LIN {X 0,Y 204.503,Z 1254.176,A -85,B 0,C 180,E1 10684.827,E2 10684.827} C_VEL
LIN {X 0,Y 208.439,Z 1245.49,A -85,B 0,C 180,E1 10678.799,E2 10678.799} C_VEL
LIN {X 0,Y 214.044,Z 1235.485,A -85,B 0,C 180,E1 10673.28,E2 10673.28} C_VEL
LIN {X 0,Y 221.45,Z 1223.468,A -85,B 0,C 180,E1 10668.071,E2 10668.071} C_VEL
LIN {X 0,Y 230.083,Z 1210.068,A -85,B 0,C 180,E1 10663.473,E2 10663.473} C_VEL
LIN {X 0,Y 239.593,Z 1195.363,A -85,B 0,C 180,E1 10659.465,E2 10659.465} C_VEL
LIN {X 0,Y 249.64,Z 1179.288,A -85,B 0,C 180,E1 10655.999,E2 10655.999} C_VEL
LIN {X 0,Y 259.481,Z 1162.559,A -85,B 0,C 180,E1 10653.172,E2 10653.172} C_VEL
LIN {X 0,Y 269.687,Z 1143.852,A -85,B 0,C 180,E1 10650.671,E2 10650.671} C_VEL
LIN {X 0,Y 279.054,Z 1124.999,A -85,B 0,C 180,E1 10648.693,E2 10648.693} C_VEL
LIN {X 0,Y 287.565,Z 1105.557,A -85,B 0,C 180,E1 10647.117,E2 10647.117} C_VEL
LIN {X 0,Y 295.468,Z 1084.875,A -85,B 0,C 180,E1 10645.827,E2 10645.827} C_VEL
LIN {X 0,Y 302.047,Z 1064.618,A -85,B 0,C 180,E1 10644.86,E2 10644.86} C_VEL
LIN {X 0,Y 307.636,Z 1042.346,A -85,B 0,C 180,E1 10644.026,E2 10644.026} C_VEL
LIN {X 0,Y 311.673,Z 1019.917,A -85,B 0,C 180,E1 10643.369,E2 10643.369} C_VEL
LIN {X 0,Y 314.482,Z 994.588,A -85,B 0,C 180,E1 10642.797,E2 10642.797} C_VEL
LIN {X 0,Y 326.356,Z 856.623,A -85,B 0,C 180,E1 10640.021,E2 10640.021} C_VEL
LIN {X 0,Y 321.509,Z 844.673,A -85,B 0,C 180,E1 10636.857,E2 10636.857} C_VEL
LIN {X 0,Y 317.747,Z 835.882,A -85,B 0,C 180,E1 10633.929,E2 10633.929} C_VEL
LIN {X 0,Y 314.507,Z 828.3,A -85,B 0,C 180,E1 10630.79,E2 10630.79} C_VEL
LIN {X 0,Y 311.943,Z 822.087,A -85,B 0,C 180,E1 10627.458,E2 10627.458} C_VEL
LIN {X 0,Y 310.729,Z 819.454,A -85,B 0,C 180,E1 10625.354,E2 10625.354} C_VEL
LIN {X 0,Y 308.92,Z 817.37,A -85,B 0,C 180,E1 10619.072,E2 10619.072} C_VEL
LIN {X 0,Y 309.517,Z 818.382,A -85,B 0,C 180,E1 10614.81,E2 10614.81} C_VEL
LIN {X 0,Y 310.912,Z 819.791,A -85,B 0,C 180,E1 10611.772,E2 10611.772} C_VEL
LIN {X 0,Y 313.909,Z 824.972,A -85,B 0,C 180,E1 10607.584,E2 10607.584} C_VEL
LIN {X 0,Y 316.917,Z 830.011,A -85,B 0,C 180,E1 10604.632,E2 10604.632} C_VEL
LIN {X 0,Y 320.006,Z 835.239,A -85,B 0,C 180,E1 10602.169,E2 10602.169} C_VEL
LIN {X 0,Y 324.529,Z 843.076,A -85,B 0,C 180,E1 10599.154,E2 10599.154} C_VEL
LIN {X 0,Y 326.398,Z 846.717,A -85,B 0,C 180,E1 10598.029,E2 10598.029} C_VEL
LIN {X 0,Y 316.958,Z 955.602,A -85,B 0,C 180,E1 10595.822,E2 10595.822} C_VEL
LIN {X 0,Y 314.556,Z 977.677,A -85,B 0,C 180,E1 10595.158,E2 10595.158} C_VEL
LIN {X 0,Y 310.815,Z 999.575,A -85,B 0,C 180,E1 10594.26,E2 10594.26} C_VEL
LIN {X 0,Y 306.147,Z 1019.787,A -85,B 0,C 180,E1 10593.187,E2 10593.187} C_VEL
LIN {X 0,Y 300.378,Z 1039.215,A -85,B 0,C 180,E1 10591.893,E2 10591.893} C_VEL
LIN {X 0,Y 293.495,Z 1058.383,A -85,B 0,C 180,E1 10590.307,E2 10590.307} C_VEL
LIN {X 0,Y 285.739,Z 1076.805,A -85,B 0,C 180,E1 10588.433,E2 10588.433} C_VEL
LIN {X 0,Y 277.363,Z 1093.945,A -85,B 0,C 180,E1 10586.278,E2 10586.278} C_VEL
LIN {X 0,Y 268.375,Z 1110.195,A -85,B 0,C 180,E1 10583.762,E2 10583.762} C_VEL
LIN {X 0,Y 259.092,Z 1125.356,A -85,B 0,C 180,E1 10580.864,E2 10580.864} C_VEL
LIN {X 0,Y 250.087,Z 1138.686,A -85,B 0,C 180,E1 10577.699,E2 10577.699} C_VEL
LIN {X 0,Y 240.767,Z 1151.437,A -85,B 0,C 180,E1 10573.908,E2 10573.908} C_VEL
LIN {X 0,Y 231.962,Z 1162.798,A -85,B 0,C 180,E1 10569.637,E2 10569.637} C_VEL
LIN {X 0,Y 223.916,Z 1172.716,A -85,B 0,C 180,E1 10564.858,E2 10564.858} C_VEL
LIN {X 0,Y 216.928,Z 1181.075,A -85,B 0,C 180,E1 10559.549,E2 10559.549} C_VEL
LIN {X 0,Y 211.256,Z 1187.948,A -85,B 0,C 180,E1 10553.721,E2 10553.721} C_VEL
LIN {X 0,Y 207.413,Z 1192.886,A -85,B 0,C 180,E1 10547.969,E2 10547.969} C_VEL
LIN {X 0,Y 204.994,Z 1196.234,A -85,B 0,C 180,E1 10542.106,E2 10542.106} C_VEL
LIN {X 0,Y 203.675,Z 1198.296,A -85,B 0,C 180,E1 10535.917,E2 10535.917} C_VEL
LIN {X 0,Y 203.338,Z 1198.982,A -85,B 0,C 180,E1 10530.282,E2 10530.282} C_VEL
LIN {X 0,Y 203.603,Z 1198.438,A -85,B 0,C 180,E1 10524.646,E2 10524.646} C_VEL
LIN {X 0,Y 204.744,Z 1196.714,A -85,B 0,C 180,E1 10518.736,E2 10518.736} C_VEL
LIN {X 0,Y 207.077,Z 1193.329,A -85,B 0,C 180,E1 10512.581,E2 10512.581} C_VEL
LIN {X 0,Y 210.986,Z 1188.339,A -85,B 0,C 180,E1 10506.543,E2 10506.543} C_VEL
LIN {X 0,Y 216.415,Z 1181.796,A -85,B 0,C 180,E1 10500.834,E2 10500.834} C_VEL
LIN {X 0,Y 223.321,Z 1173.527,A -85,B 0,C 180,E1 10495.469,E2 10495.469} C_VEL
LIN {X 0,Y 231.054,Z 1164.004,A -85,B 0,C 180,E1 10490.769,E2 10490.769} C_VEL
LIN {X 0,Y 240.16,Z 1152.37,A -85,B 0,C 180,E1 10486.284,E2 10486.284} C_VEL
LIN {X 0,Y 249.432,Z 1139.816,A -85,B 0,C 180,E1 10482.477,E2 10482.477} C_VEL
LIN {X 0,Y 258.967,Z 1125.723,A -85,B 0,C 180,E1 10479.102,E2 10479.102} C_VEL
LIN {X 0,Y 268.247,Z 1110.632,A -85,B 0,C 180,E1 10476.201,E2 10476.201} C_VEL
LIN {X 0,Y 277.137,Z 1094.668,A -85,B 0,C 180,E1 10473.711,E2 10473.711} C_VEL
LIN {X 0,Y 285.608,Z 1077.369,A -85,B 0,C 180,E1 10471.524,E2 10471.524} C_VEL
LIN {X 0,Y 293.368,Z 1059.066,A -85,B 0,C 180,E1 10469.65,E2 10469.65} C_VEL
LIN {X 0,Y 300.496,Z 1039.32,A -85,B 0,C 180,E1 10468.01,E2 10468.01} C_VEL
LIN {X 0,Y 306.179,Z 1020.196,A -85,B 0,C 180,E1 10466.733,E2 10466.733} C_VEL
LIN {X 0,Y 311.012,Z 999.341,A -85,B 0,C 180,E1 10465.626,E2 10465.626} C_VEL
LIN {X 0,Y 314.792,Z 977.037,A -85,B 0,C 180,E1 10464.718,E2 10464.718} C_VEL
LIN {X 0,Y 317.162,Z 954.96,A -85,B 0,C 180,E1 10464.06,E2 10464.06} C_VEL
LIN {X 0,Y 326.534,Z 846.621,A -85,B 0,C 180,E1 10461.851,E2 10461.851} C_VEL
LIN {X 0,Y 321.954,Z 838.389,A -85,B 0,C 180,E1 10458.985,E2 10458.985} C_VEL
LIN {X 0,Y 318.029,Z 831.737,A -85,B 0,C 180,E1 10456.062,E2 10456.062} C_VEL
LIN {X 0,Y 315.638,Z 827.791,A -85,B 0,C 180,E1 10453.931,E2 10453.931} C_VEL
LIN {X 0,Y 313.48,Z 824.081,A -85,B 0,C 180,E1 10451.592,E2 10451.592} C_VEL
LIN {X 0,Y 312.025,Z 822.099,A -85,B 0,C 180,E1 10449.716,E2 10449.716} C_VEL
LIN {X 0,Y 311.103,Z 821.621,A -85,B 0,C 180,E1 10448.407,E2 10448.407} C_VEL
LIN {X 0,Y 309.694,Z 823.43,A -85,B 0,C 180,E1 10446.383,E2 10446.383} C_VEL
LIN {X 0,Y 308.511,Z 825.827,A -85,B 0,C 180,E1 10444.02,E2 10444.02} C_VEL
LIN {X 0,Y 308.312,Z 825.919,A -85,B 0,C 180,E1 10443.183,E2 10443.183} C_VEL
LIN {X 0,Y 308.242,Z 825.769,A -85,B 0,C 180,E1 10439.814,E2 10439.814} C_VEL
LIN {X 0,Y 309.952,Z 827.753,A -85,B 0,C 180,E1 10434.632,E2 10434.632} C_VEL
LIN {X 0,Y 311.302,Z 831.115,A -85,B 0,C 180,E1 10432.248,E2 10432.248} C_VEL
LIN {X 0,Y 313.701,Z 836.931,A -85,B 0,C 180,E1 10429.161,E2 10429.161} C_VEL
LIN {X 0,Y 317.548,Z 846.48,A -85,B 0,C 180,E1 10425.457,E2 10425.457} C_VEL
LIN {X 0,Y 321.377,Z 856.081,A -85,B 0,C 180,E1 10422.529,E2 10422.529} C_VEL
LIN {X 0,Y 323.306,Z 861.466,A -85,B 0,C 180,E1 10421.198,E2 10421.198} C_VEL
LIN {X 0,Y 309.794,Z 1010.819,A -85,B 0,C 180,E1 10418.218,E2 10418.218} C_VEL
LIN {X 0,Y 306.147,Z 1033.255,A -85,B 0,C 180,E1 10417.618,E2 10417.618} C_VEL
LIN {X 0,Y 300.877,Z 1055.874,A -85,B 0,C 180,E1 10416.851,E2 10416.851} C_VEL
LIN {X 0,Y 294.479,Z 1076.961,A -85,B 0,C 180,E1 10415.956,E2 10415.956} C_VEL
LIN {X 0,Y 286.773,Z 1097.528,A -85,B 0,C 180,E1 10414.812,E2 10414.812} C_VEL
LIN {X 0,Y 278.03,Z 1117.659,A -85,B 0,C 180,E1 10413.333,E2 10413.333} C_VEL
LIN {X 0,Y 268.525,Z 1137.044,A -85,B 0,C 180,E1 10411.489,E2 10411.489} C_VEL
LIN {X 0,Y 258.368,Z 1155.588,A -85,B 0,C 180,E1 10409.215,E2 10409.215} C_VEL
LIN {X 0,Y 248.104,Z 1172.667,A -85,B 0,C 180,E1 10406.531,E2 10406.531} C_VEL
LIN {X 0,Y 237.325,Z 1189.476,A -85,B 0,C 180,E1 10403.173,E2 10403.173} C_VEL
LIN {X 0,Y 227.365,Z 1204.365,A -85,B 0,C 180,E1 10399.395,E2 10399.395} C_VEL
LIN {X 0,Y 217.967,Z 1218.039,A -85,B 0,C 180,E1 10394.943,E2 10394.943} C_VEL
LIN {X 0,Y 209.514,Z 1230.606,A -85,B 0,C 180,E1 10389.752,E2 10389.752} C_VEL
LIN {X 0,Y 202.783,Z 1241.437,A -85,B 0,C 180,E1 10384.071,E2 10384.071} C_VEL
LIN {X 0,Y 197.975,Z 1250.46,A -85,B 0,C 180,E1 10378.013,E2 10378.013} C_VEL
LIN {X 0,Y 195.11,Z 1257.789,A -85,B 0,C 180,E1 10371.651,E2 10371.651} C_VEL
LIN {X 0,Y 194.074,Z 1263.415,A -85,B 0,C 180,E1 10365.233,E2 10365.233} C_VEL
LIN {X 0,Y 194.355,Z 1266.89,A -85,B 0,C 180,E1 10359.475,E2 10359.475} C_VEL
LIN {X 0,Y 195.05,Z 1268.792,A -85,B 0,C 180,E1 10354.41,E2 10354.41} C_VEL
LIN {X 0,Y 195.396,Z 1269.368,A -85,B 0,C 180,E1 10350,E2 10350} C_VEL
LIN {X 0,Y 195.051,Z 1268.784,A -85,B 0,C 180,E1 10345.59,E2 10345.59} C_VEL
LIN {X 0,Y 194.358,Z 1266.876,A -85,B 0,C 180,E1 10340.525,E2 10340.525} C_VEL
LIN {X 0,Y 194.075,Z 1263.395,A -85,B 0,C 180,E1 10334.767,E2 10334.767} C_VEL
LIN {X 0,Y 195.111,Z 1257.763,A -85,B 0,C 180,E1 10328.349,E2 10328.349} C_VEL
LIN {X 0,Y 197.976,Z 1250.423,A -85,B 0,C 180,E1 10321.987,E2 10321.987} C_VEL
LIN {X 0,Y 202.888,Z 1241.215,A -85,B 0,C 180,E1 10315.82,E2 10315.82} C_VEL
LIN {X 0,Y 209.622,Z 1230.376,A -85,B 0,C 180,E1 10310.169,E2 10310.169} C_VEL
LIN {X 0,Y 218.43,Z 1217.266,A -85,B 0,C 180,E1 10304.807,E2 10304.807} C_VEL
LIN {X 0,Y 227.549,Z 1203.98,A -85,B 0,C 180,E1 10300.523,E2 10300.523} C_VEL
LIN {X 0,Y 237.811,Z 1188.63,A -85,B 0,C 180,E1 10296.657,E2 10296.657} C_VEL
LIN {X 0,Y 248.097,Z 1172.525,A -85,B 0,C 180,E1 10293.467,E2 10293.467} C_VEL
LIN {X 0,Y 258.358,Z 1155.409,A -85,B 0,C 180,E1 10290.782,E2 10290.782} C_VEL
LIN {X 0,Y 268.135,Z 1137.555,A -85,B 0,C 180,E1 10288.587,E2 10288.587} C_VEL
LIN {X 0,Y 277.633,Z 1118.248,A -85,B 0,C 180,E1 10286.733,E2 10286.733} C_VEL
LIN {X 0,Y 286.322,Z 1098.341,A -85,B 0,C 180,E1 10285.255,E2 10285.255} C_VEL
LIN {X 0,Y 294.117,Z 1077.571,A -85,B 0,C 180,E1 10284.089,E2 10284.089} C_VEL
LIN {X 0,Y 300.513,Z 1056.674,A -85,B 0,C 180,E1 10283.193,E2 10283.193} C_VEL
LIN {X 0,Y 305.922,Z 1033.657,A -85,B 0,C 180,E1 10282.406,E2 10282.406} C_VEL
LIN {X 0,Y 309.597,Z 1011.199,A -85,B 0,C 180,E1 10281.803,E2 10281.803} C_VEL
LIN {X 0,Y 321.287,Z 881.947,A -85,B 0,C 180,E1 10279.213,E2 10279.213} C_VEL
LIN {X 0,Y 323.122,Z 860.936,A -85,B 0,C 180,E1 10278.772,E2 10278.772} C_VEL
LIN {X 0,Y 318.787,Z 849.865,A -85,B 0,C 180,E1 10275.695,E2 10275.695} C_VEL
LIN {X 0,Y 315.749,Z 842.456,A -85,B 0,C 180,E1 10273.132,E2 10273.132} C_VEL
LIN {X 0,Y 312.944,Z 835.521,A -85,B 0,C 180,E1 10270.214,E2 10270.214} C_VEL
LIN {X 0,Y 310.65,Z 829.666,A -85,B 0,C 180,E1 10267.025,E2 10267.025} C_VEL
LIN {X 0,Y 309.548,Z 827.277,A -85,B 0,C 180,E1 10265.003,E2 10265.003} C_VEL
LIN {X 0,Y 307.943,Z 825.297,A -85,B 0,C 180,E1 10258.883,E2 10258.883} C_VEL
LIN {X 0,Y 308.882,Z 826.716,A -85,B 0,C 180,E1 10253.868,E2 10253.868} C_VEL
LIN {X 0,Y 309.825,Z 827.75,A -85,B 0,C 180,E1 10251.93,E2 10251.93} C_VEL
LIN {X 0,Y 312.678,Z 832.844,A -85,B 0,C 180,E1 10247.816,E2 10247.816} C_VEL
LIN {X 0,Y 315.421,Z 837.566,A -85,B 0,C 180,E1 10245.028,E2 10245.028} C_VEL
LIN {X 0,Y 319.312,Z 844.257,A -85,B 0,C 180,E1 10241.893,E2 10241.893} C_VEL
LIN {X 0,Y 323.211,Z 851.495,A -85,B 0,C 180,E1 10239.265,E2 10239.265} C_VEL
LIN {X 0,Y 313.851,Z 956.436,A -85,B 0,C 180,E1 10237.152,E2 10237.152} C_VEL
LIN {X 0,Y 311.402,Z 978.497,A -85,B 0,C 180,E1 10236.496,E2 10236.496} C_VEL
LIN {X 0,Y 307.529,Z 1000.715,A -85,B 0,C 180,E1 10235.595,E2 10235.595} C_VEL
LIN {X 0,Y 302.837,Z 1020.632,A -85,B 0,C 180,E1 10234.552,E2 10234.552} C_VEL
LIN {X 0,Y 296.748,Z 1040.612,A -85,B 0,C 180,E1 10233.235,E2 10233.235} C_VEL
LIN {X 0,Y 289.672,Z 1059.779,A -85,B 0,C 180,E1 10231.661,E2 10231.661} C_VEL
LIN {X 0,Y 281.69,Z 1078.201,A -85,B 0,C 180,E1 10229.8,E2 10229.8} C_VEL
LIN {X 0,Y 272.902,Z 1095.643,A -85,B 0,C 180,E1 10227.616,E2 10227.616} C_VEL
LIN {X 0,Y 263.781,Z 1111.586,A -85,B 0,C 180,E1 10225.149,E2 10225.149} C_VEL
LIN {X 0,Y 254.167,Z 1126.757,A -85,B 0,C 180,E1 10222.249,E2 10222.249} C_VEL
LIN {X 0,Y 244.817,Z 1140.088,A -85,B 0,C 180,E1 10219.072,E2 10219.072} C_VEL
LIN {X 0,Y 235.107,Z 1152.841,A -85,B 0,C 180,E1 10215.251,E2 10215.251} C_VEL
LIN {X 0,Y 225.891,Z 1164.204,A -85,B 0,C 180,E1 10210.925,E2 10210.925} C_VEL
LIN {X 0,Y 217.427,Z 1174.123,A -85,B 0,C 180,E1 10206.058,E2 10206.058} C_VEL
LIN {X 0,Y 210.035,Z 1182.482,A -85,B 0,C 180,E1 10200.621,E2 10200.621} C_VEL
LIN {X 0,Y 203.992,Z 1189.354,A -85,B 0,C 180,E1 10194.621,E2 10194.621} C_VEL
LIN {X 0,Y 199.876,Z 1194.288,A -85,B 0,C 180,E1 10188.672,E2 10188.672} C_VEL
LIN {X 0,Y 197.258,Z 1197.632,A -85,B 0,C 180,E1 10182.589,E2 10182.589} C_VEL
LIN {X 0,Y 195.826,Z 1199.688,A -85,B 0,C 180,E1 10176.155,E2 10176.155} C_VEL
LIN {X 0,Y 195.461,Z 1200.373,A -85,B 0,C 180,E1 10170.293,E2 10170.293} C_VEL
LIN {X 0,Y 195.749,Z 1199.829,A -85,B 0,C 180,E1 10164.431,E2 10164.431} C_VEL
LIN {X 0,Y 196.987,Z 1198.11,A -85,B 0,C 180,E1 10158.286,E2 10158.286} C_VEL
LIN {X 0,Y 199.511,Z 1194.73,A -85,B 0,C 180,E1 10151.898,E2 10151.898} C_VEL
LIN {X 0,Y 203.706,Z 1189.743,A -85,B 0,C 180,E1 10145.651,E2 10145.651} C_VEL
LIN {X 0,Y 209.345,Z 1183.378,A -85,B 0,C 180,E1 10139.902,E2 10139.902} C_VEL
LIN {X 0,Y 216.567,Z 1175.187,A -85,B 0,C 180,E1 10134.429,E2 10134.429} C_VEL
LIN {X 0,Y 224.875,Z 1165.489,A -85,B 0,C 180,E1 10129.523,E2 10129.523} C_VEL
LIN {X 0,Y 234.479,Z 1153.771,A -85,B 0,C 180,E1 10124.941,E2 10124.941} C_VEL
LIN {X 0,Y 244.143,Z 1141.214,A -85,B 0,C 180,E1 10121.103,E2 10121.103} C_VEL
LIN {X 0,Y 254.043,Z 1127.119,A -85,B 0,C 180,E1 10117.715,E2 10117.715} C_VEL
LIN {X 0,Y 263.651,Z 1112.025,A -85,B 0,C 180,E1 10114.813,E2 10114.813} C_VEL
LIN {X 0,Y 272.698,Z 1096.316,A -85,B 0,C 180,E1 10112.366,E2 10112.366} C_VEL
LIN {X 0,Y 281.564,Z 1078.757,A -85,B 0,C 180,E1 10110.156,E2 10110.156} C_VEL
LIN {X 0,Y 289.549,Z 1060.452,A -85,B 0,C 180,E1 10108.294,E2 10108.294} C_VEL
LIN {X 0,Y 296.635,Z 1041.453,A -85,B 0,C 180,E1 10106.722,E2 10106.722} C_VEL
LIN {X 0,Y 302.716,Z 1021.58,A -85,B 0,C 180,E1 10105.401,E2 10105.401} C_VEL
LIN {X 0,Y 307.685,Z 1000.721,A -85,B 0,C 180,E1 10104.302,E2 10104.302} C_VEL
LIN {X 0,Y 311.574,Z 978.414,A -85,B 0,C 180,E1 10103.399,E2 10103.399} C_VEL
LIN {X 0,Y 314.022,Z 956.329,A -85,B 0,C 180,E1 10102.743,E2 10102.743} C_VEL
LIN {X 0,Y 323.31,Z 851.467,A -85,B 0,C 180,E1 10100.597,E2 10100.597} C_VEL
LIN {X 0,Y 319.054,Z 843.692,A -85,B 0,C 180,E1 10097.697,E2 10097.697} C_VEL
LIN {X 0,Y 315.502,Z 837.537,A -85,B 0,C 180,E1 10094.781,E2 10094.781} C_VEL
LIN {X 0,Y 312.197,Z 831.799,A -85,B 0,C 180,E1 10091.266,E2 10091.266} C_VEL
LIN {X 0,Y 309.761,Z 827.402,A -85,B 0,C 180,E1 10087.419,E2 10087.419} C_VEL
LIN {X 0,Y 308.312,Z 825.919,A -85,B 0,C 180,E1 10083.183,E2 10083.183} C_VEL
LIN {X 0,Y 308.071,Z 826.562,A -85,B 0,C 180,E1 10081.851,E2 10081.851} C_VEL
LIN {X 0,Y 307.707,Z 830.18,A -85,B 0,C 180,E1 10079.77,E2 10079.77} C_VEL
LIN {X 0,Y 307.754,Z 834.066,A -85,B 0,C 180,E1 10077.574,E2 10077.574} C_VEL
LIN {X 0,Y 307.988,Z 834.719,A -85,B 0,C 180,E1 10076.748,E2 10076.748} C_VEL
LIN {X 0,Y 308.868,Z 835.69,A -85,B 0,C 180,E1 10074.8,E2 10074.8} C_VEL
LIN {X 0,Y 310.059,Z 838.814,A -85,B 0,C 180,E1 10072.589,E2 10072.589} C_VEL
LIN {X 0,Y 312.272,Z 844.511,A -85,B 0,C 180,E1 10069.578,E2 10069.578} C_VEL
LIN {X 0,Y 315.763,Z 853.626,A -85,B 0,C 180,E1 10066.029,E2 10066.029} C_VEL
LIN {X 0,Y 319.367,Z 863.118,A -85,B 0,C 180,E1 10063.12,E2 10063.12} C_VEL
LIN {X 0,Y 320.243,Z 865.843,A -85,B 0,C 180,E1 10062.46,E2 10062.46} C_VEL
LIN {X 0,Y 306.873,Z 1009.439,A -85,B 0,C 180,E1 10059.624,E2 10059.624} C_VEL
LIN {X 0,Y 303.144,Z 1031.872,A -85,B 0,C 180,E1 10059.035,E2 10059.035} C_VEL
LIN {X 0,Y 297.613,Z 1055.051,A -85,B 0,C 180,E1 10058.263,E2 10058.263} C_VEL
LIN {X 0,Y 291.047,Z 1076.14,A -85,B 0,C 180,E1 10057.384,E2 10057.384} C_VEL
LIN {X 0,Y 283.113,Z 1096.815,A -85,B 0,C 180,E1 10056.259,E2 10056.259} C_VEL
LIN {X 0,Y 274.051,Z 1117.051,A -85,B 0,C 180,E1 10054.794,E2 10054.794} C_VEL
LIN {X 0,Y 264.54,Z 1135.858,A -85,B 0,C 180,E1 10053.029,E2 10053.029} C_VEL
LIN {X 0,Y 254.108,Z 1154.319,A -85,B 0,C 180,E1 10050.797,E2 10050.797} C_VEL
LIN {X 0,Y 243.602,Z 1171.198,A -85,B 0,C 180,E1 10048.168,E2 10048.168} C_VEL
LIN {X 0,Y 232.395,Z 1187.998,A -85,B 0,C 180,E1 10044.829,E2 10044.829} C_VEL
LIN {X 0,Y 222.179,Z 1202.598,A -85,B 0,C 180,E1 10041.125,E2 10041.125} C_VEL
LIN {X 0,Y 212.561,Z 1215.854,A -85,B 0,C 180,E1 10036.809,E2 10036.809} C_VEL
LIN {X 0,Y 203.49,Z 1228.54,A -85,B 0,C 180,E1 10031.553,E2 10031.553} C_VEL
LIN {X 0,Y 196.282,Z 1239.311,A -85,B 0,C 180,E1 10025.859,E2 10025.859} C_VEL
LIN {X 0,Y 190.815,Z 1248.57,A -85,B 0,C 180,E1 10019.508,E2 10019.508} C_VEL
LIN {X 0,Y 187.422,Z 1256.269,A -85,B 0,C 180,E1 10012.645,E2 10012.645} C_VEL
LIN {X 0,Y 186.158,Z 1261.965,A -85,B 0,C 180,E1 10005.897,E2 10005.897} C_VEL
LIN {X 0,Y 186.395,Z 1265.465,A -85,B 0,C 180,E1 9999.884,E2 9999.884} C_VEL
LIN {X 0,Y 187.128,Z 1267.39,A -85,B 0,C 180,E1 9994.597,E2 9994.597} C_VEL
LIN {X 0,Y 187.517,Z 1267.978,A -85,B 0,C 180,E1 9990,E2 9990} C_VEL
LIN {X 0,Y 187.129,Z 1267.382,A -85,B 0,C 180,E1 9985.403,E2 9985.403} C_VEL
LIN {X 0,Y 186.397,Z 1265.451,A -85,B 0,C 180,E1 9980.116,E2 9980.116} C_VEL
LIN {X 0,Y 186.165,Z 1261.892,A -85,B 0,C 180,E1 9974.021,E2 9974.021} C_VEL
LIN {X 0,Y 187.425,Z 1256.24,A -85,B 0,C 180,E1 9967.353,E2 9967.353} C_VEL
LIN {X 0,Y 190.815,Z 1248.53,A -85,B 0,C 180,E1 9960.492,E2 9960.492} C_VEL
LIN {X 0,Y 196.374,Z 1239.116,A -85,B 0,C 180,E1 9954.053,E2 9954.053} C_VEL
LIN {X 0,Y 203.899,Z 1227.901,A -85,B 0,C 180,E1 9948.173,E2 9948.173} C_VEL
LIN {X 0,Y 213.053,Z 1215.077,A -85,B 0,C 180,E1 9942.939,E2 9942.939} C_VEL
LIN {X 0,Y 222.974,Z 1201.339,A -85,B 0,C 180,E1 9938.557,E2 9938.557} C_VEL
LIN {X 0,Y 233.655,Z 1186.075,A -85,B 0,C 180,E1 9934.757,E2 9934.757} C_VEL
LIN {X 0,Y 244.282,Z 1169.981,A -85,B 0,C 180,E1 9931.644,E2 9931.644} C_VEL
LIN {X 0,Y 255.67,Z 1151.401,A -85,B 0,C 180,E1 9928.839,E2 9928.839} C_VEL
LIN {X 0,Y 265.833,Z 1133.253,A -85,B 0,C 180,E1 9926.714,E2 9926.714} C_VEL
LIN {X 0,Y 275.331,Z 1114.112,A -85,B 0,C 180,E1 9924.984,E2 9924.984} C_VEL
LIN {X 0,Y 284.178,Z 1093.822,A -85,B 0,C 180,E1 9923.577,E2 9923.577} C_VEL
LIN {X 0,Y 291.704,Z 1073.828,A -85,B 0,C 180,E1 9922.524,E2 9922.524} C_VEL
LIN {X 0,Y 298.327,Z 1051.97,A -85,B 0,C 180,E1 9921.633,E2 9921.633} C_VEL
LIN {X 0,Y 303.385,Z 1029.836,A -85,B 0,C 180,E1 9920.918,E2 9920.918} C_VEL
LIN {X 0,Y 307.012,Z 1006.706,A -85,B 0,C 180,E1 9920.33,E2 9920.33} C_VEL
LIN {X 0,Y 320.098,Z 865.479,A -85,B 0,C 180,E1 9917.543,E2 9917.543} C_VEL
LIN {X 0,Y 316.451,Z 855.814,A -85,B 0,C 180,E1 9914.735,E2 9914.735} C_VEL
LIN {X 0,Y 313.905,Z 849.247,A -85,B 0,C 180,E1 9912.415,E2 9912.415} C_VEL
LIN {X 0,Y 311.398,Z 842.697,A -85,B 0,C 180,E1 9909.611,E2 9909.611} C_VEL
LIN {X 0,Y 309.321,Z 837.129,A -85,B 0,C 180,E1 9906.496,E2 9906.496} C_VEL
LIN {X 0,Y 308.476,Z 835.166,A -85,B 0,C 180,E1 9904.834,E2 9904.834} C_VEL
LIN {X 0,Y 306.968,Z 833.238,A -85,B 0,C 180,E1 9898.88,E2 9898.88} C_VEL
LIN {X 0,Y 307.987,Z 834.758,A -85,B 0,C 180,E1 9893.663,E2 9893.663} C_VEL
LIN {X 0,Y 308.74,Z 835.704,A -85,B 0,C 180,E1 9892.089,E2 9892.089} C_VEL
LIN {X 0,Y 311.379,Z 840.551,A -85,B 0,C 180,E1 9888.14,E2 9888.14} C_VEL
LIN {X 0,Y 313.94,Z 845.121,A -85,B 0,C 180,E1 9885.427,E2 9885.427} C_VEL
LIN {X 0,Y 317.591,Z 851.642,A -85,B 0,C 180,E1 9882.361,E2 9882.361} C_VEL
LIN {X 0,Y 320.145,Z 856.609,A -85,B 0,C 180,E1 9880.519,E2 9880.519} C_VEL
LIN {X 0,Y 310.931,Z 957.084,A -85,B 0,C 180,E1 9878.513,E2 9878.513} C_VEL
LIN {X 0,Y 308.435,Z 979.222,A -85,B 0,C 180,E1 9877.864,E2 9877.864} C_VEL
LIN {X 0,Y 304.425,Z 1001.803,A -85,B 0,C 180,E1 9876.961,E2 9876.961} C_VEL
LIN {X 0,Y 299.536,Z 1022.031,A -85,B 0,C 180,E1 9875.912,E2 9875.912} C_VEL
LIN {X 0,Y 293.285,Z 1042.009,A -85,B 0,C 180,E1 9874.609,E2 9874.609} C_VEL
LIN {X 0,Y 286.016,Z 1061.175,A -85,B 0,C 180,E1 9873.05,E2 9873.05} C_VEL
LIN {X 0,Y 278.163,Z 1078.893,A -85,B 0,C 180,E1 9871.286,E2 9871.286} C_VEL
LIN {X 0,Y 269.096,Z 1096.403,A -85,B 0,C 180,E1 9869.124,E2 9869.124} C_VEL
LIN {X 0,Y 259.304,Z 1113.046,A -85,B 0,C 180,E1 9866.573,E2 9866.573} C_VEL
LIN {X 0,Y 249.395,Z 1128.157,A -85,B 0,C 180,E1 9863.689,E2 9863.689} C_VEL
LIN {X 0,Y 239.695,Z 1141.491,A -85,B 0,C 180,E1 9860.505,E2 9860.505} C_VEL
LIN {X 0,Y 229.583,Z 1154.245,A -85,B 0,C 180,E1 9856.659,E2 9856.659} C_VEL
LIN {X 0,Y 219.937,Z 1165.611,A -85,B 0,C 180,E1 9852.284,E2 9852.284} C_VEL
LIN {X 0,Y 211.042,Z 1175.53,A -85,B 0,C 180,E1 9847.33,E2 9847.33} C_VEL
LIN {X 0,Y 203.222,Z 1183.889,A -85,B 0,C 180,E1 9841.764,E2 9841.764} C_VEL
LIN {X 0,Y 196.782,Z 1190.76,A -85,B 0,C 180,E1 9835.587,E2 9835.587} C_VEL
LIN {X 0,Y 192.37,Z 1195.69,A -85,B 0,C 180,E1 9829.429,E2 9829.429} C_VEL
LIN {X 0,Y 189.44,Z 1199.166,A -85,B 0,C 180,E1 9822.807,E2 9822.807} C_VEL
LIN {X 0,Y 187.982,Z 1201.081,A -85,B 0,C 180,E1 9816.413,E2 9816.413} C_VEL
LIN {X 0,Y 187.583,Z 1201.763,A -85,B 0,C 180,E1 9810.305,E2 9810.305} C_VEL
LIN {X 0,Y 187.899,Z 1201.222,A -85,B 0,C 180,E1 9804.197,E2 9804.197} C_VEL
LIN {X 0,Y 189.241,Z 1199.507,A -85,B 0,C 180,E1 9797.799,E2 9797.799} C_VEL
LIN {X 0,Y 191.98,Z 1196.131,A -85,B 0,C 180,E1 9791.162,E2 9791.162} C_VEL
LIN {X 0,Y 196.479,Z 1191.147,A -85,B 0,C 180,E1 9784.694,E2 9784.694} C_VEL
LIN {X 0,Y 202.49,Z 1184.783,A -85,B 0,C 180,E1 9778.771,E2 9778.771} C_VEL
LIN {X 0,Y 210.136,Z 1176.591,A -85,B 0,C 180,E1 9773.165,E2 9773.165} C_VEL
LIN {X 0,Y 218.882,Z 1166.891,A -85,B 0,C 180,E1 9768.171,E2 9768.171} C_VEL
LIN {X 0,Y 228.933,Z 1155.172,A -85,B 0,C 180,E1 9763.533,E2 9763.533} C_VEL
LIN {X 0,Y 239,Z 1142.612,A -85,B 0,C 180,E1 9759.669,E2 9759.669} C_VEL
LIN {X 0,Y 249.274,Z 1128.514,A -85,B 0,C 180,E1 9756.274,E2 9756.274} C_VEL
LIN {X 0,Y 259.214,Z 1113.418,A -85,B 0,C 180,E1 9753.377,E2 9753.377} C_VEL
LIN {X 0,Y 268.977,Z 1096.908,A -85,B 0,C 180,E1 9750.834,E2 9750.834} C_VEL
LIN {X 0,Y 278.04,Z 1079.44,A -85,B 0,C 180,E1 9748.667,E2 9748.667} C_VEL
LIN {X 0,Y 286.26,Z 1060.97,A -85,B 0,C 180,E1 9746.825,E2 9746.825} C_VEL
LIN {X 0,Y 293.905,Z 1040.648,A -85,B 0,C 180,E1 9745.19,E2 9745.19} C_VEL
LIN {X 0,Y 299.979,Z 1021.05,A -85,B 0,C 180,E1 9743.926,E2 9743.926} C_VEL
LIN {X 0,Y 305.031,Z 999.773,A -85,B 0,C 180,E1 9742.843,E2 9742.843} C_VEL
LIN {X 0,Y 308.766,Z 978.042,A -85,B 0,C 180,E1 9741.995,E2 9741.995} C_VEL
LIN {X 0,Y 311.314,Z 954.493,A -85,B 0,C 180,E1 9741.321,E2 9741.321} C_VEL
LIN {X 0,Y 320.308,Z 856.643,A -85,B 0,C 180,E1 9739.375,E2 9739.375} C_VEL
LIN {X 0,Y 316.455,Z 849.501,A -85,B 0,C 180,E1 9736.521,E2 9736.521} C_VEL
LIN {X 0,Y 313.032,Z 843.311,A -85,B 0,C 180,E1 9733.39,E2 9733.39} C_VEL
LIN {X 0,Y 310.778,Z 839.337,A -85,B 0,C 180,E1 9730.755,E2 9730.755} C_VEL
LIN {X 0,Y 308.598,Z 835.224,A -85,B 0,C 180,E1 9727.073,E2 9727.073} C_VEL
LIN {X 0,Y 307.197,Z 833.534,A -85,B 0,C 180,E1 9721.306,E2 9721.306} C_VEL
LIN {X 0,Y 307.988,Z 834.719,A -85,B 0,C 180,E1 9716.748,E2 9716.748} C_VEL
LIN {X 0,Y 308.381,Z 836.177,A -85,B 0,C 180,E1 9715.548,E2 9715.548} C_VEL
LIN {X 0,Y 308.782,Z 840.188,A -85,B 0,C 180,E1 9714.067,E2 9714.067} C_VEL
LIN {X 0,Y 309.737,Z 848.626,A -85,B 0,C 180,E1 9711.557,E2 9711.557} C_VEL
LIN {X 0,Y 310.244,Z 850.455,A -85,B 0,C 180,E1 9710.791,E2 9710.791} C_VEL
LIN {X 0,Y 313.234,Z 858.526,A -85,B 0,C 180,E1 9707.37,E2 9707.37} C_VEL
LIN {X 0,Y 316.665,Z 868.171,A -85,B 0,C 180,E1 9704.291,E2 9704.291} C_VEL
LIN {X 0,Y 317.334,Z 870.262,A -85,B 0,C 180,E1 9703.744,E2 9703.744} C_VEL
LIN {X 0,Y 304.142,Z 1008.043,A -85,B 0,C 180,E1 9701.056,E2 9701.056} C_VEL
LIN {X 0,Y 300.337,Z 1030.453,A -85,B 0,C 180,E1 9700.48,E2 9700.48} C_VEL
LIN {X 0,Y 294.706,Z 1053.629,A -85,B 0,C 180,E1 9699.728,E2 9699.728} C_VEL
LIN {X 0,Y 288.274,Z 1074.055,A -85,B 0,C 180,E1 9698.904,E2 9698.904} C_VEL
LIN {X 0,Y 280.186,Z 1094.768,A -85,B 0,C 180,E1 9697.821,E2 9697.821} C_VEL
LIN {X 0,Y 271.074,Z 1114.778,A -85,B 0,C 180,E1 9696.429,E2 9696.429} C_VEL
LIN {X 0,Y 261.453,Z 1133.451,A -85,B 0,C 180,E1 9694.743,E2 9694.743} C_VEL
LIN {X 0,Y 251.032,Z 1151.398,A -85,B 0,C 180,E1 9692.645,E2 9692.645} C_VEL
LIN {X 0,Y 239.679,Z 1169.171,A -85,B 0,C 180,E1 9689.961,E2 9689.961} C_VEL
LIN {X 0,Y 228.325,Z 1185.619,A -85,B 0,C 180,E1 9686.76,E2 9686.76} C_VEL
LIN {X 0,Y 217.6,Z 1200.288,A -85,B 0,C 180,E1 9683.082,E2 9683.082} C_VEL
LIN {X 0,Y 207.397,Z 1213.67,A -85,B 0,C 180,E1 9678.768,E2 9678.768} C_VEL
LIN {X 0,Y 197.688,Z 1226.477,A -85,B 0,C 180,E1 9673.459,E2 9673.459} C_VEL
LIN {X 0,Y 189.848,Z 1237.33,A -85,B 0,C 180,E1 9667.655,E2 9667.655} C_VEL
LIN {X 0,Y 183.785,Z 1246.678,A -85,B 0,C 180,E1 9661.119,E2 9661.119} C_VEL
LIN {X 0,Y 179.862,Z 1254.544,A -85,B 0,C 180,E1 9653.941,E2 9653.941} C_VEL
LIN {X 0,Y 178.292,Z 1260.307,A -85,B 0,C 180,E1 9646.954,E2 9646.954} C_VEL
LIN {X 0,Y 178.399,Z 1263.886,A -85,B 0,C 180,E1 9640.658,E2 9640.658} C_VEL
LIN {X 0,Y 179.158,Z 1265.895,A -85,B 0,C 180,E1 9635.123,E2 9635.123} C_VEL
LIN {X 0,Y 179.621,Z 1266.544,A -85,B 0,C 180,E1 9630.638,E2 9630.638} C_VEL
LIN {X 0,Y 179.345,Z 1266.197,A -85,B 0,C 180,E1 9626.164,E2 9626.164} C_VEL
LIN {X 0,Y 178.538,Z 1264.475,A -85,B 0,C 180,E1 9620.654,E2 9620.654} C_VEL
LIN {X 0,Y 178.203,Z 1261.323,A -85,B 0,C 180,E1 9614.71,E2 9614.71} C_VEL
LIN {X 0,Y 179.407,Z 1255.747,A -85,B 0,C 180,E1 9607.385,E2 9607.385} C_VEL
LIN {X 0,Y 182.666,Z 1248.656,A -85,B 0,C 180,E1 9600.487,E2 9600.487} C_VEL
LIN {X 0,Y 188.2,Z 1239.617,A -85,B 0,C 180,E1 9593.855,E2 9593.855} C_VEL
LIN {X 0,Y 195.956,Z 1228.706,A -85,B 0,C 180,E1 9587.662,E2 9587.662} C_VEL
LIN {X 0,Y 204.81,Z 1217.061,A -85,B 0,C 180,E1 9582.512,E2 9582.512} C_VEL
LIN {X 0,Y 215.269,Z 1203.249,A -85,B 0,C 180,E1 9577.813,E2 9577.813} C_VEL
LIN {X 0,Y 226.354,Z 1188.201,A -85,B 0,C 180,E1 9573.859,E2 9573.859} C_VEL
LIN {X 0,Y 237.372,Z 1172.499,A -85,B 0,C 180,E1 9570.642,E2 9570.642} C_VEL
LIN {X 0,Y 248.03,Z 1156.091,A -85,B 0,C 180,E1 9568.017,E2 9568.017} C_VEL
LIN {X 0,Y 258.697,Z 1138.078,A -85,B 0,C 180,E1 9565.774,E2 9565.774} C_VEL
LIN {X 0,Y 268.626,Z 1119.513,A -85,B 0,C 180,E1 9563.971,E2 9563.971} C_VEL
LIN {X 0,Y 277.665,Z 1100.293,A -85,B 0,C 180,E1 9562.539,E2 9562.539} C_VEL
LIN {X 0,Y 285.69,Z 1080.552,A -85,B 0,C 180,E1 9561.422,E2 9561.422} C_VEL
LIN {X 0,Y 292.986,Z 1059.117,A -85,B 0,C 180,E1 9560.488,E2 9560.488} C_VEL
LIN {X 0,Y 298.823,Z 1036.922,A -85,B 0,C 180,E1 9559.721,E2 9559.721} C_VEL
LIN {X 0,Y 302.97,Z 1014.751,A -85,B 0,C 180,E1 9559.116,E2 9559.116} C_VEL
LIN {X 0,Y 306.279,Z 985.823,A -85,B 0,C 180,E1 9558.501,E2 9558.501} C_VEL
LIN {X 0,Y 317.165,Z 869.887,A -85,B 0,C 180,E1 9556.247,E2 9556.247} C_VEL
LIN {X 0,Y 313.689,Z 860.215,A -85,B 0,C 180,E1 9553.267,E2 9553.267} C_VEL
LIN {X 0,Y 310.45,Z 851.308,A -85,B 0,C 180,E1 9549.734,E2 9549.734} C_VEL
LIN {X 0,Y 308.223,Z 845.041,A -85,B 0,C 180,E1 9546.332,E2 9546.332} C_VEL
LIN {X 0,Y 307.405,Z 843.055,A -85,B 0,C 180,E1 9544.664,E2 9544.664} C_VEL
LIN {X 0,Y 305.993,Z 841.179,A -85,B 0,C 180,E1 9538.876,E2 9538.876} C_VEL
LIN {X 0,Y 307.096,Z 842.801,A -85,B 0,C 180,E1 9533.456,E2 9533.456} C_VEL
LIN {X 0,Y 307.659,Z 843.649,A -85,B 0,C 180,E1 9532.249,E2 9532.249} C_VEL
LIN {X 0,Y 310.09,Z 848.257,A -85,B 0,C 180,E1 9528.468,E2 9528.468} C_VEL
LIN {X 0,Y 312.565,Z 852.855,A -85,B 0,C 180,E1 9525.74,E2 9525.74} C_VEL
LIN {X 0,Y 315.947,Z 859.143,A -85,B 0,C 180,E1 9522.789,E2 9522.789} C_VEL
LIN {X 0,Y 317.223,Z 861.85,A -85,B 0,C 180,E1 9521.794,E2 9521.794} C_VEL
LIN {X 0,Y 308.179,Z 957.865,A -85,B 0,C 180,E1 9519.896,E2 9519.896} C_VEL
LIN {X 0,Y 305.595,Z 980.312,A -85,B 0,C 180,E1 9519.245,E2 9519.245} C_VEL
LIN {X 0,Y 301.439,Z 1003.159,A -85,B 0,C 180,E1 9518.342,E2 9518.342} C_VEL
LIN {X 0,Y 296.408,Z 1023.429,A -85,B 0,C 180,E1 9517.302,E2 9517.302} C_VEL
LIN {X 0,Y 289.995,Z 1043.406,A -85,B 0,C 180,E1 9516.015,E2 9516.015} C_VEL
LIN {X 0,Y 282.531,Z 1062.571,A -85,B 0,C 180,E1 9514.475,E2 9514.475} C_VEL
LIN {X 0,Y 274.461,Z 1080.289,A -85,B 0,C 180,E1 9512.731,E2 9512.731} C_VEL
LIN {X 0,Y 265.13,Z 1097.801,A -85,B 0,C 180,E1 9510.589,E2 9510.589} C_VEL
LIN {X 0,Y 255.407,Z 1113.865,A -85,B 0,C 180,E1 9508.155,E2 9508.155} C_VEL
LIN {X 0,Y 245.438,Z 1128.686,A -85,B 0,C 180,E1 9505.374,E2 9505.374} C_VEL
LIN {X 0,Y 234.729,Z 1142.894,A -85,B 0,C 180,E1 9502,E2 9502} C_VEL
LIN {X 0,Y 224.206,Z 1155.649,A -85,B 0,C 180,E1 9498.135,E2 9498.135} C_VEL
LIN {X 0,Y 214.116,Z 1167.017,A -85,B 0,C 180,E1 9493.717,E2 9493.717} C_VEL
LIN {X 0,Y 204.767,Z 1176.937,A -85,B 0,C 180,E1 9488.682,E2 9488.682} C_VEL
LIN {X 0,Y 196.495,Z 1185.296,A -85,B 0,C 180,E1 9482.987,E2 9482.987} C_VEL
LIN {X 0,Y 189.632,Z 1192.166,A -85,B 0,C 180,E1 9476.626,E2 9476.626} C_VEL
LIN {X 0,Y 184.902,Z 1197.092,A -85,B 0,C 180,E1 9470.247,E2 9470.247} C_VEL
LIN {X 0,Y 181.725,Z 1200.565,A -85,B 0,C 180,E1 9463.361,E2 9463.361} C_VEL
LIN {X 0,Y 180.142,Z 1202.474,A -85,B 0,C 180,E1 9456.693,E2 9456.693} C_VEL
LIN {X 0,Y 179.704,Z 1203.153,A -85,B 0,C 180,E1 9450.319,E2 9450.319} C_VEL
LIN {X 0,Y 180.05,Z 1202.614,A -85,B 0,C 180,E1 9443.944,E2 9443.944} C_VEL
LIN {X 0,Y 181.509,Z 1200.904,A -85,B 0,C 180,E1 9437.271,E2 9437.271} C_VEL
LIN {X 0,Y 184.483,Z 1197.531,A -85,B 0,C 180,E1 9430.366,E2 9430.366} C_VEL
LIN {X 0,Y 189.31,Z 1192.552,A -85,B 0,C 180,E1 9423.664,E2 9423.664} C_VEL
LIN {X 0,Y 195.722,Z 1186.188,A -85,B 0,C 180,E1 9417.562,E2 9417.562} C_VEL
LIN {X 0,Y 203.816,Z 1177.996,A -85,B 0,C 180,E1 9411.823,E2 9411.823} C_VEL
LIN {X 0,Y 213.016,Z 1168.294,A -85,B 0,C 180,E1 9406.743,E2 9406.743} C_VEL
LIN {X 0,Y 223.534,Z 1156.572,A -85,B 0,C 180,E1 9402.056,E2 9402.056} C_VEL
LIN {X 0,Y 234.014,Z 1144.01,A -85,B 0,C 180,E1 9398.173,E2 9398.173} C_VEL
LIN {X 0,Y 244.67,Z 1129.91,A -85,B 0,C 180,E1 9394.777,E2 9394.777} C_VEL
LIN {X 0,Y 254.857,Z 1114.951,A -85,B 0,C 180,E1 9391.916,E2 9391.916} C_VEL
LIN {X 0,Y 264.665,Z 1098.934,A -85,B 0,C 180,E1 9389.453,E2 9389.453} C_VEL
LIN {X 0,Y 273.976,Z 1081.533,A -85,B 0,C 180,E1 9387.301,E2 9387.301} C_VEL
LIN {X 0,Y 282.417,Z 1063.223,A -85,B 0,C 180,E1 9385.476,E2 9385.476} C_VEL
LIN {X 0,Y 289.89,Z 1044.22,A -85,B 0,C 180,E1 9383.939,E2 9383.939} C_VEL
LIN {X 0,Y 296.299,Z 1024.343,A -85,B 0,C 180,E1 9382.647,E2 9382.647} C_VEL
LIN {X 0,Y 301.525,Z 1003.545,A -85,B 0,C 180,E1 9381.574,E2 9381.574} C_VEL
LIN {X 0,Y 305.63,Z 981.302,A -85,B 0,C 180,E1 9380.687,E2 9380.687} C_VEL
LIN {X 0,Y 308.234,Z 959.318,A -85,B 0,C 180,E1 9380.038,E2 9380.038} C_VEL
LIN {X 0,Y 314.756,Z 889.383,A -85,B 0,C 180,E1 9378.626,E2 9378.626} C_VEL
LIN {X 0,Y 317.377,Z 861.724,A -85,B 0,C 180,E1 9378.078,E2 9378.078} C_VEL
LIN {X 0,Y 313.502,Z 854.385,A -85,B 0,C 180,E1 9374.877,E2 9374.877} C_VEL
LIN {X 0,Y 311.273,Z 850.331,A -85,B 0,C 180,E1 9372.617,E2 9372.617} C_VEL
LIN {X 0,Y 309.522,Z 847.049,A -85,B 0,C 180,E1 9370.422,E2 9370.422} C_VEL
LIN {X 0,Y 307.536,Z 843.115,A -85,B 0,C 180,E1 9366.909,E2 9366.909} C_VEL
LIN {X 0,Y 306.222,Z 841.479,A -85,B 0,C 180,E1 9361.123,E2 9361.123} C_VEL
LIN {X 0,Y 307.674,Z 843.247,A -85,B 0,C 180,E1 9355.247,E2 9355.247} C_VEL
LIN {X 0,Y 308.827,Z 846.511,A -85,B 0,C 180,E1 9352.933,E2 9352.933} C_VEL
LIN {X 0,Y 310.244,Z 850.455,A -85,B 0,C 180,E1 9350.791,E2 9350.791} C_VEL
LIN {X 0,Y 311.002,Z 853.48,A -85,B 0,C 180,E1 9349.709,E2 9349.709} C_VEL
LIN {X 0,Y 311.872,Z 859.853,A -85,B 0,C 180,E1 9348.29,E2 9348.29} C_VEL
LIN {X 0,Y 313.394,Z 870.6,A -85,B 0,C 180,E1 9346.171,E2 9346.171} C_VEL
LIN {X 0,Y 313.896,Z 872.538,A -85,B 0,C 180,E1 9345.671,E2 9345.671} C_VEL
LIN {X 0,Y 314.561,Z 874.93,A -85,B 0,C 180,E1 9345.048,E2 9345.048} C_VEL
LIN {X 0,Y 301.593,Z 1006.741,A -85,B 0,C 180,E1 9342.512,E2 9342.512} C_VEL
LIN {X 0,Y 297.706,Z 1029.126,A -85,B 0,C 180,E1 9341.95,E2 9341.95} C_VEL
LIN {X 0,Y 292.038,Z 1052.059,A -85,B 0,C 180,E1 9341.227,E2 9341.227} C_VEL
LIN {X 0,Y 285.457,Z 1072.631,A -85,B 0,C 180,E1 9340.422,E2 9340.422} C_VEL
LIN {X 0,Y 277.218,Z 1093.339,A -85,B 0,C 180,E1 9339.378,E2 9339.378} C_VEL
LIN {X 0,Y 267.907,Z 1113.339,A -85,B 0,C 180,E1 9338.033,E2 9338.033} C_VEL
LIN {X 0,Y 258.154,Z 1131.826,A -85,B 0,C 180,E1 9336.414,E2 9336.414} C_VEL
LIN {X 0,Y 247.338,Z 1149.941,A -85,B 0,C 180,E1 9334.348,E2 9334.348} C_VEL
LIN {X 0,Y 235.972,Z 1167.195,A -85,B 0,C 180,E1 9331.801,E2 9331.801} C_VEL
LIN {X 0,Y 224.528,Z 1183.241,A -85,B 0,C 180,E1 9328.757,E2 9328.757} C_VEL
LIN {X 0,Y 213.254,Z 1198.016,A -85,B 0,C 180,E1 9325.11,E2 9325.11} C_VEL
LIN {X 0,Y 202.419,Z 1211.592,A -85,B 0,C 180,E1 9320.783,E2 9320.783} C_VEL
LIN {X 0,Y 192.589,Z 1223.837,A -85,B 0,C 180,E1 9315.76,E2 9315.76} C_VEL
LIN {X 0,Y 183.986,Z 1234.804,A -85,B 0,C 180,E1 9309.885,E2 9309.885} C_VEL
LIN {X 0,Y 177.162,Z 1244.37,A -85,B 0,C 180,E1 9303.191,E2 9303.191} C_VEL
LIN {X 0,Y 172.707,Z 1252.142,A -85,B 0,C 180,E1 9296.102,E2 9296.102} C_VEL
LIN {X 0,Y 170.554,Z 1258.106,A -85,B 0,C 180,E1 9288.809,E2 9288.809} C_VEL
LIN {X 0,Y 170.393,Z 1262.303,A -85,B 0,C 180,E1 9281.496,E2 9281.496} C_VEL
LIN {X 0,Y 171.105,Z 1264.297,A -85,B 0,C 180,E1 9276.038,E2 9276.038} C_VEL
LIN {X 0,Y 171.687,Z 1265.065,A -85,B 0,C 180,E1 9271.669,E2 9271.669} C_VEL
LIN {X 0,Y 171.661,Z 1265.03,A -85,B 0,C 180,E1 9267.997,E2 9267.997} C_VEL
LIN {X 0,Y 171.045,Z 1264.18,A -85,B 0,C 180,E1 9263.586,E2 9263.586} C_VEL
LIN {X 0,Y 170.338,Z 1261.971,A -85,B 0,C 180,E1 9257.801,E2 9257.801} C_VEL
LIN {X 0,Y 170.671,Z 1257.564,A -85,B 0,C 180,E1 9250.493,E2 9250.493} C_VEL
LIN {X 0,Y 173.023,Z 1251.486,A -85,B 0,C 180,E1 9243.209,E2 9243.209} C_VEL
LIN {X 0,Y 177.708,Z 1243.501,A -85,B 0,C 180,E1 9236.152,E2 9236.152} C_VEL
LIN {X 0,Y 184.755,Z 1233.704,A -85,B 0,C 180,E1 9229.504,E2 9229.504} C_VEL
LIN {X 0,Y 193.551,Z 1222.56,A -85,B 0,C 180,E1 9223.681,E2 9223.681} C_VEL
LIN {X 0,Y 204.121,Z 1209.43,A -85,B 0,C 180,E1 9218.468,E2 9218.468} C_VEL
LIN {X 0,Y 215.187,Z 1195.376,A -85,B 0,C 180,E1 9214.204,E2 9214.204} C_VEL
LIN {X 0,Y 227.106,Z 1179.545,A -85,B 0,C 180,E1 9210.501,E2 9210.501} C_VEL
LIN {X 0,Y 238.947,Z 1162.757,A -85,B 0,C 180,E1 9207.492,E2 9207.492} C_VEL
LIN {X 0,Y 249.677,Z 1145.94,A -85,B 0,C 180,E1 9205.175,E2 9205.175} C_VEL
LIN {X 0,Y 260.885,Z 1126.549,A -85,B 0,C 180,E1 9203.105,E2 9203.105} C_VEL
LIN {X 0,Y 270.421,Z 1108.053,A -85,B 0,C 180,E1 9201.586,E2 9201.586} C_VEL
LIN {X 0,Y 278.934,Z 1088.893,A -85,B 0,C 180,E1 9200.391,E2 9200.391} C_VEL
LIN {X 0,Y 287.194,Z 1067.042,A -85,B 0,C 180,E1 9199.361,E2 9199.361} C_VEL
LIN {X 0,Y 293.724,Z 1045.48,A -85,B 0,C 180,E1 9198.557,E2 9198.557} C_VEL
LIN {X 0,Y 298.724,Z 1023.257,A -85,B 0,C 180,E1 9197.901,E2 9197.901} C_VEL
LIN {X 0,Y 302.124,Z 1000.655,A -85,B 0,C 180,E1 9197.373,E2 9197.373} C_VEL
LIN {X 0,Y 314.376,Z 874.467,A -85,B 0,C 180,E1 9194.928,E2 9194.928} C_VEL
LIN {X 0,Y 311.236,Z 865.2,A -85,B 0,C 180,E1 9191.911,E2 9191.911} C_VEL
LIN {X 0,Y 308.663,Z 857.777,A -85,B 0,C 180,E1 9188.757,E2 9188.757} C_VEL
LIN {X 0,Y 306.882,Z 852.387,A -85,B 0,C 180,E1 9185.703,E2 9185.703} C_VEL
LIN {X 0,Y 306.248,Z 850.875,A -85,B 0,C 180,E1 9184.306,E2 9184.306} C_VEL
LIN {X 0,Y 305.019,Z 849.113,A -85,B 0,C 180,E1 9178.685,E2 9178.685} C_VEL
LIN {X 0,Y 306.389,Z 850.992,A -85,B 0,C 180,E1 9172.876,E2 9172.876} C_VEL
LIN {X 0,Y 308.812,Z 855.962,A -85,B 0,C 180,E1 9168.798,E2 9168.798} C_VEL
LIN {X 0,Y 311.2,Z 860.586,A -85,B 0,C 180,E1 9166.056,E2 9166.056} C_VEL
LIN {X 0,Y 314.472,Z 866.965,A -85,B 0,C 180,E1 9163.095,E2 9163.095} C_VEL
LIN {X 0,Y 305.604,Z 958.707,A -85,B 0,C 180,E1 9161.302,E2 9161.302} C_VEL
LIN {X 0,Y 302.936,Z 981.403,A -85,B 0,C 180,E1 9160.651,E2 9160.651} C_VEL
LIN {X 0,Y 298.75,Z 1003.989,A -85,B 0,C 180,E1 9159.773,E2 9159.773} C_VEL
LIN {X 0,Y 293.459,Z 1024.828,A -85,B 0,C 180,E1 9158.721,E2 9158.721} C_VEL
LIN {X 0,Y 286.883,Z 1044.803,A -85,B 0,C 180,E1 9157.452,E2 9157.452} C_VEL
LIN {X 0,Y 278.973,Z 1064.544,A -85,B 0,C 180,E1 9155.884,E2 9155.884} C_VEL
LIN {X 0,Y 270.187,Z 1083.095,A -85,B 0,C 180,E1 9154.056,E2 9154.056} C_VEL
LIN {X 0,Y 260.621,Z 1100.473,A -85,B 0,C 180,E1 9151.928,E2 9151.928} C_VEL
LIN {X 0,Y 250.623,Z 1116.318,A -85,B 0,C 180,E1 9149.508,E2 9149.508} C_VEL
LIN {X 0,Y 239.682,Z 1131.831,A -85,B 0,C 180,E1 9146.542,E2 9146.542} C_VEL
LIN {X 0,Y 228.68,Z 1145.879,A -85,B 0,C 180,E1 9143.14,E2 9143.14} C_VEL
LIN {X 0,Y 217.822,Z 1158.356,A -85,B 0,C 180,E1 9139.233,E2 9139.233} C_VEL
LIN {X 0,Y 207.391,Z 1169.477,A -85,B 0,C 180,E1 9134.738,E2 9134.738} C_VEL
LIN {X 0,Y 197.705,Z 1179.22,A -85,B 0,C 180,E1 9129.584,E2 9129.584} C_VEL
LIN {X 0,Y 189.122,Z 1187.432,A -85,B 0,C 180,E1 9123.718,E2 9123.718} C_VEL
LIN {X 0,Y 182.266,Z 1193.839,A -85,B 0,C 180,E1 9117.438,E2 9117.438} C_VEL
LIN {X 0,Y 177.065,Z 1198.849,A -85,B 0,C 180,E1 9110.493,E2 9110.493} C_VEL
LIN {X 0,Y 173.811,Z 1202.236,A -85,B 0,C 180,E1 9103.303,E2 9103.303} C_VEL
LIN {X 0,Y 172.211,Z 1203.979,A -85,B 0,C 180,E1 9096.333,E2 9096.333} C_VEL
LIN {X 0,Y 171.826,Z 1204.553,A -85,B 0,C 180,E1 9089.667,E2 9089.667} C_VEL
LIN {X 0,Y 172.296,Z 1203.895,A -85,B 0,C 180,E1 9083,E2 9083} C_VEL
LIN {X 0,Y 174.117,Z 1201.893,A -85,B 0,C 180,E1 9075.705,E2 9075.705} C_VEL
LIN {X 0,Y 177.628,Z 1198.401,A -85,B 0,C 180,E1 9068.539,E2 9068.539} C_VEL
LIN {X 0,Y 183.073,Z 1193.154,A -85,B 0,C 180,E1 9061.632,E2 9061.632} C_VEL
LIN {X 0,Y 190.545,Z 1186.133,A -85,B 0,C 180,E1 9055.114,E2 9055.114} C_VEL
LIN {X 0,Y 198.978,Z 1178.075,A -85,B 0,C 180,E1 9049.594,E2 9049.594} C_VEL
LIN {X 0,Y 208.86,Z 1168.117,A -85,B 0,C 180,E1 9044.498,E2 9044.498} C_VEL
LIN {X 0,Y 218.875,Z 1157.32,A -85,B 0,C 180,E1 9040.283,E2 9040.283} C_VEL
LIN {X 0,Y 229.82,Z 1144.615,A -85,B 0,C 180,E1 9036.405,E2 9036.405} C_VEL
LIN {X 0,Y 240.238,Z 1131.305,A -85,B 0,C 180,E1 9033.225,E2 9033.225} C_VEL
LIN {X 0,Y 250.966,Z 1116.041,A -85,B 0,C 180,E1 9030.33,E2 9030.33} C_VEL
LIN {X 0,Y 261.4,Z 1099.391,A -85,B 0,C 180,E1 9027.818,E2 9027.818} C_VEL
LIN {X 0,Y 270.825,Z 1082.216,A -85,B 0,C 180,E1 9025.737,E2 9025.737} C_VEL
LIN {X 0,Y 279.499,Z 1063.741,A -85,B 0,C 180,E1 9023.939,E2 9023.939} C_VEL
LIN {X 0,Y 287.551,Z 1043.415,A -85,B 0,C 180,E1 9022.348,E2 9022.348} C_VEL
LIN {X 0,Y 294.094,Z 1023.242,A -85,B 0,C 180,E1 9021.086,E2 9021.086} C_VEL
LIN {X 0,Y 299.383,Z 1002.005,A -85,B 0,C 180,E1 9020.036,E2 9020.036} C_VEL
LIN {X 0,Y 303.271,Z 980.365,A -85,B 0,C 180,E1 9019.214,E2 9019.214} C_VEL
LIN {X 0,Y 306.029,Z 955.996,A -85,B 0,C 180,E1 9018.532,E2 9018.532} C_VEL
LIN {X 0,Y 314.597,Z 866.992,A -85,B 0,C 180,E1 9016.764,E2 9016.764} C_VEL
LIN {X 0,Y 311.383,Z 860.733,A -85,B 0,C 180,E1 9013.841,E2 9013.841} C_VEL
LIN {X 0,Y 308.617,Z 855.21,A -85,B 0,C 180,E1 9010.548,E2 9010.548} C_VEL
LIN {X 0,Y 306.476,Z 851.006,A -85,B 0,C 180,E1 9006.745,E2 9006.745} C_VEL
LIN {X 0,Y 305.247,Z 849.419,A -85,B 0,C 180,E1 9001.126,E2 9001.126} C_VEL
LIN {X 0,Y 306.563,Z 851.074,A -85,B 0,C 180,E1 8995.511,E2 8995.511} C_VEL
LIN {X 0,Y 307.657,Z 854.366,A -85,B 0,C 180,E1 8993.188,E2 8993.188} C_VEL
LIN {X 0,Y 309.605,Z 860.087,A -85,B 0,C 180,E1 8990.239,E2 8990.239} C_VEL
LIN {X 0,Y 312.29,Z 867.915,A -85,B 0,C 180,E1 8987.19,E2 8987.19} C_VEL
LIN {X 0,Y 313.896,Z 872.538,A -85,B 0,C 180,E1 8985.671,E2 8985.671} C_VEL
LIN {X 0,Y 314.067,Z 874.595,A -85,B 0,C 180,E1 8985.389,E2 8985.389} C_VEL
LIN {X 0,Y 313.78,Z 877.976,A -85,B 0,C 180,E1 8985.296,E2 8985.296} C_VEL
LIN {X 0,Y 312.688,Z 883.798,A -85,B 0,C 180,E1 8985.522,E2 8985.522} C_VEL
LIN {X 0,Y 310.753,Z 892.768,A -85,B 0,C 180,E1 8986.05,E2 8986.05} C_VEL
LIN {X 0,Y 310.289,Z 896.165,A -85,B 0,C 180,E1 8986.071,E2 8986.071} C_VEL
LIN {X 0,Y 299.216,Z 1005.655,A -85,B 0,C 180,E1 8983.987,E2 8983.987} C_VEL
LIN {X 0,Y 295.204,Z 1028.143,A -85,B 0,C 180,E1 8983.434,E2 8983.434} C_VEL
LIN {X 0,Y 289.442,Z 1050.934,A -85,B 0,C 180,E1 8982.736,E2 8982.736} C_VEL
LIN {X 0,Y 282.399,Z 1072.355,A -85,B 0,C 180,E1 8981.919,E2 8981.919} C_VEL
LIN {X 0,Y 274.46,Z 1091.91,A -85,B 0,C 180,E1 8980.967,E2 8980.967} C_VEL
LIN {X 0,Y 265,Z 1111.818,A -85,B 0,C 180,E1 8979.679,E2 8979.679} C_VEL
LIN {X 0,Y 254.868,Z 1130.555,A -85,B 0,C 180,E1 8978.09,E2 8978.09} C_VEL
LIN {X 0,Y 243.873,Z 1148.486,A -85,B 0,C 180,E1 8976.1,E2 8976.1} C_VEL
LIN {X 0,Y 231.937,Z 1166.037,A -85,B 0,C 180,E1 8973.56,E2 8973.56} C_VEL
LIN {X 0,Y 219.588,Z 1182.667,A -85,B 0,C 180,E1 8970.419,E2 8970.419} C_VEL
LIN {X 0,Y 207.74,Z 1197.565,A -85,B 0,C 180,E1 8966.724,E2 8966.724} C_VEL
LIN {X 0,Y 196.439,Z 1210.998,A -85,B 0,C 180,E1 8962.354,E2 8962.354} C_VEL
LIN {X 0,Y 185.218,Z 1224.15,A -85,B 0,C 180,E1 8956.72,E2 8956.72} C_VEL
LIN {X 0,Y 176.118,Z 1235.156,A -85,B 0,C 180,E1 8950.471,E2 8950.471} C_VEL
LIN {X 0,Y 169.043,Z 1244.533,A -85,B 0,C 180,E1 8943.371,E2 8943.371} C_VEL
LIN {X 0,Y 164.581,Z 1251.908,A -85,B 0,C 180,E1 8935.938,E2 8935.938} C_VEL
LIN {X 0,Y 162.528,Z 1257.605,A -85,B 0,C 180,E1 8928.285,E2 8928.285} C_VEL
LIN {X 0,Y 162.483,Z 1261.173,A -85,B 0,C 180,E1 8921.356,E2 8921.356} C_VEL
LIN {X 0,Y 163.321,Z 1263.173,A -85,B 0,C 180,E1 8915.269,E2 8915.269} C_VEL
LIN {X 0,Y 163.858,Z 1263.763,A -85,B 0,C 180,E1 8910.699,E2 8910.699} C_VEL
LIN {X 0,Y 163.608,Z 1263.482,A -85,B 0,C 180,E1 8906.496,E2 8906.496} C_VEL
LIN {X 0,Y 162.676,Z 1261.923,A -85,B 0,C 180,E1 8900.448,E2 8900.448} C_VEL
LIN {X 0,Y 162.377,Z 1258.628,A -85,B 0,C 180,E1 8893.546,E2 8893.546} C_VEL
LIN {X 0,Y 163.879,Z 1253.422,A -85,B 0,C 180,E1 8885.873,E2 8885.873} C_VEL
LIN {X 0,Y 167.75,Z 1246.411,A -85,B 0,C 180,E1 8878.365,E2 8878.365} C_VEL
LIN {X 0,Y 174.113,Z 1237.579,A -85,B 0,C 180,E1 8871.25,E2 8871.25} C_VEL
LIN {X 0,Y 182.867,Z 1226.871,A -85,B 0,C 180,E1 8864.702,E2 8864.702} C_VEL
LIN {X 0,Y 193.226,Z 1214.74,A -85,B 0,C 180,E1 8859.09,E2 8859.09} C_VEL
LIN {X 0,Y 204.045,Z 1201.865,A -85,B 0,C 180,E1 8854.593,E2 8854.593} C_VEL
LIN {X 0,Y 216.755,Z 1186.138,A -85,B 0,C 180,E1 8850.393,E2 8850.393} C_VEL
LIN {X 0,Y 228.746,Z 1170.364,A -85,B 0,C 180,E1 8847.192,E2 8847.192} C_VEL
LIN {X 0,Y 240.681,Z 1153.156,A -85,B 0,C 180,E1 8844.528,E2 8844.528} C_VEL
LIN {X 0,Y 252.005,Z 1135.09,A -85,B 0,C 180,E1 8842.388,E2 8842.388} C_VEL
LIN {X 0,Y 262.818,Z 1115.778,A -85,B 0,C 180,E1 8840.635,E2 8840.635} C_VEL
LIN {X 0,Y 272.41,Z 1096.187,A -85,B 0,C 180,E1 8839.289,E2 8839.289} C_VEL
LIN {X 0,Y 280.755,Z 1076.165,A -85,B 0,C 180,E1 8838.264,E2 8838.264} C_VEL
LIN {X 0,Y 288.371,Z 1053.985,A -85,B 0,C 180,E1 8837.382,E2 8837.382} C_VEL
LIN {X 0,Y 294.29,Z 1031.724,A -85,B 0,C 180,E1 8836.674,E2 8836.674} C_VEL
LIN {X 0,Y 298.478,Z 1009.225,A -85,B 0,C 180,E1 8836.106,E2 8836.106} C_VEL
LIN {X 0,Y 302.112,Z 976.85,A -85,B 0,C 180,E1 8835.458,E2 8835.458} C_VEL
LIN {X 0,Y 311.763,Z 879.008,A -85,B 0,C 180,E1 8833.588,E2 8833.588} C_VEL
LIN {X 0,Y 309.236,Z 871.33,A -85,B 0,C 180,E1 8830.903,E2 8830.903} C_VEL
LIN {X 0,Y 307.142,Z 864.768,A -85,B 0,C 180,E1 8828.046,E2 8828.046} C_VEL
LIN {X 0,Y 305.58,Z 859.722,A -85,B 0,C 180,E1 8825.068,E2 8825.068} C_VEL
LIN {X 0,Y 305.186,Z 858.764,A -85,B 0,C 180,E1 8824.133,E2 8824.133} C_VEL
LIN {X 0,Y 304.044,Z 857.054,A -85,B 0,C 180,E1 8818.681,E2 8818.681} C_VEL
LIN {X 0,Y 305.323,Z 858.911,A -85,B 0,C 180,E1 8813.04,E2 8813.04} C_VEL
LIN {X 0,Y 307.609,Z 863.82,A -85,B 0,C 180,E1 8809.038,E2 8809.038} C_VEL
LIN {X 0,Y 309.845,Z 868.315,A -85,B 0,C 180,E1 8806.375,E2 8806.375} C_VEL
LIN {X 0,Y 311.837,Z 872.583,A -85,B 0,C 180,E1 8804.409,E2 8804.409} C_VEL
LIN {X 0,Y 303.211,Z 959.607,A -85,B 0,C 180,E1 8802.729,E2 8802.729} C_VEL
LIN {X 0,Y 300.462,Z 982.493,A -85,B 0,C 180,E1 8802.081,E2 8802.081} C_VEL
LIN {X 0,Y 296.291,Z 1004.651,A -85,B 0,C 180,E1 8801.237,E2 8801.237} C_VEL
LIN {X 0,Y 290.893,Z 1025.592,A -85,B 0,C 180,E1 8800.204,E2 8800.204} C_VEL
LIN {X 0,Y 284.233,Z 1045.431,A -85,B 0,C 180,E1 8798.973,E2 8798.973} C_VEL
LIN {X 0,Y 276.102,Z 1065.374,A -85,B 0,C 180,E1 8797.427,E2 8797.427} C_VEL
LIN {X 0,Y 267.254,Z 1083.716,A -85,B 0,C 180,E1 8795.665,E2 8795.665} C_VEL
LIN {X 0,Y 257.371,Z 1101.233,A -85,B 0,C 180,E1 8793.565,E2 8793.565} C_VEL
LIN {X 0,Y 246.705,Z 1117.717,A -85,B 0,C 180,E1 8791.091,E2 8791.091} C_VEL
LIN {X 0,Y 235.407,Z 1133.232,A -85,B 0,C 180,E1 8788.151,E2 8788.151} C_VEL
LIN {X 0,Y 224.011,Z 1147.281,A -85,B 0,C 180,E1 8784.764,E2 8784.764} C_VEL
LIN {X 0,Y 212.72,Z 1159.76,A -85,B 0,C 180,E1 8780.853,E2 8780.853} C_VEL
LIN {X 0,Y 201.815,Z 1170.883,A -85,B 0,C 180,E1 8776.328,E2 8776.328} C_VEL
LIN {X 0,Y 191.636,Z 1180.627,A -85,B 0,C 180,E1 8771.101,E2 8771.101} C_VEL
LIN {X 0,Y 182.55,Z 1188.839,A -85,B 0,C 180,E1 8765.106,E2 8765.106} C_VEL
LIN {X 0,Y 175.238,Z 1195.245,A -85,B 0,C 180,E1 8758.637,E2 8758.637} C_VEL
LIN {X 0,Y 169.572,Z 1200.316,A -85,B 0,C 180,E1 8751.309,E2 8751.309} C_VEL
LIN {X 0,Y 166.113,Z 1203.634,A -85,B 0,C 180,E1 8743.931,E2 8743.931} C_VEL
LIN {X 0,Y 164.371,Z 1205.372,A -85,B 0,C 180,E1 8736.637,E2 8736.637} C_VEL
LIN {X 0,Y 163.948,Z 1205.943,A -85,B 0,C 180,E1 8729.651,E2 8729.651} C_VEL
LIN {X 0,Y 164.465,Z 1205.288,A -85,B 0,C 180,E1 8722.665,E2 8722.665} C_VEL
LIN {X 0,Y 166.446,Z 1203.292,A -85,B 0,C 180,E1 8715.031,E2 8715.031} C_VEL
LIN {X 0,Y 170.253,Z 1199.803,A -85,B 0,C 180,E1 8707.56,E2 8707.56} C_VEL
LIN {X 0,Y 176.104,Z 1194.559,A -85,B 0,C 180,E1 8700.4,E2 8700.4} C_VEL
LIN {X 0,Y 184.061,Z 1187.539,A -85,B 0,C 180,E1 8693.694,E2 8693.694} C_VEL
LIN {X 0,Y 192.984,Z 1179.478,A -85,B 0,C 180,E1 8688.062,E2 8688.062} C_VEL
LIN {X 0,Y 203.361,Z 1169.52,A -85,B 0,C 180,E1 8682.898,E2 8682.898} C_VEL
LIN {X 0,Y 214.434,Z 1158.068,A -85,B 0,C 180,E1 8678.434,E2 8678.434} C_VEL
LIN {X 0,Y 226.26,Z 1144.73,A -85,B 0,C 180,E1 8674.447,E2 8674.447} C_VEL
LIN {X 0,Y 237.661,Z 1130.564,A -85,B 0,C 180,E1 8671.163,E2 8671.163} C_VEL
LIN {X 0,Y 248.772,Z 1114.961,A -85,B 0,C 180,E1 8668.337,E2 8668.337} C_VEL
LIN {X 0,Y 259.133,Z 1098.525,A -85,B 0,C 180,E1 8665.973,E2 8665.973} C_VEL
LIN {X 0,Y 268.647,Z 1081.38,A -85,B 0,C 180,E1 8663.981,E2 8663.981} C_VEL
LIN {X 0,Y 277.22,Z 1063.304,A -85,B 0,C 180,E1 8662.29,E2 8662.29} C_VEL
LIN {X 0,Y 285.044,Z 1043.703,A -85,B 0,C 180,E1 8660.807,E2 8660.807} C_VEL
LIN {X 0,Y 291.588,Z 1023.761,A -85,B 0,C 180,E1 8659.594,E2 8659.594} C_VEL
LIN {X 0,Y 296.949,Z 1002.645,A -85,B 0,C 180,E1 8658.574,E2 8658.574} C_VEL
LIN {X 0,Y 300.845,Z 981.217,A -85,B 0,C 180,E1 8657.776,E2 8657.776} C_VEL
LIN {X 0,Y 303.824,Z 955.044,A -85,B 0,C 180,E1 8657.064,E2 8657.064} C_VEL
LIN {X 0,Y 312.024,Z 872.509,A -85,B 0,C 180,E1 8655.477,E2 8655.477} C_VEL
LIN {X 0,Y 308.973,Z 866.26,A -85,B 0,C 180,E1 8652.333,E2 8652.333} C_VEL
LIN {X 0,Y 307.041,Z 862.471,A -85,B 0,C 180,E1 8649.749,E2 8649.749} C_VEL
LIN {X 0,Y 305.336,Z 858.825,A -85,B 0,C 180,E1 8646.393,E2 8646.393} C_VEL
LIN {X 0,Y 304.272,Z 857.36,A -85,B 0,C 180,E1 8641.13,E2 8641.13} C_VEL
LIN {X 0,Y 305.496,Z 858.99,A -85,B 0,C 180,E1 8635.683,E2 8635.683} C_VEL
LIN {X 0,Y 306.493,Z 862.217,A -85,B 0,C 180,E1 8633.444,E2 8633.444} C_VEL
LIN {X 0,Y 308.389,Z 868.178,A -85,B 0,C 180,E1 8630.436,E2 8630.436} C_VEL
LIN {X 0,Y 310.687,Z 875.333,A -85,B 0,C 180,E1 8627.69,E2 8627.69} C_VEL
LIN {X 0,Y 311.958,Z 879.533,A -85,B 0,C 180,E1 8626.377,E2 8626.377} C_VEL
LIN {X 0,Y 310.289,Z 896.165,A -85,B 0,C 180,E1 8626.071,E2 8626.071} C_VEL
LIN {X 0,Y 309.265,Z 903.858,A -85,B 0,C 180,E1 8626.103,E2 8626.103} C_VEL
LIN {X 0,Y 305.597,Z 924.399,A -85,B 0,C 180,E1 8626.854,E2 8626.854} C_VEL
LIN {X 0,Y 304.735,Z 931.004,A -85,B 0,C 180,E1 8626.872,E2 8626.872} C_VEL
LIN {X 0,Y 297.001,Z 1004.847,A -85,B 0,C 180,E1 8625.479,E2 8625.479} C_VEL
LIN {X 0,Y 292.828,Z 1027.516,A -85,B 0,C 180,E1 8624.935,E2 8624.935} C_VEL
LIN {X 0,Y 287.184,Z 1049.362,A -85,B 0,C 180,E1 8624.287,E2 8624.287} C_VEL
LIN {X 0,Y 280.441,Z 1069.784,A -85,B 0,C 180,E1 8623.544,E2 8623.544} C_VEL
LIN {X 0,Y 272.363,Z 1089.458,A -85,B 0,C 180,E1 8622.639,E2 8622.639} C_VEL
LIN {X 0,Y 262.665,Z 1109.631,A -85,B 0,C 180,E1 8621.408,E2 8621.408} C_VEL
LIN {X 0,Y 252.339,Z 1128.417,A -85,B 0,C 180,E1 8619.893,E2 8619.893} C_VEL
LIN {X 0,Y 241.053,Z 1146.397,A -85,B 0,C 180,E1 8617.975,E2 8617.975} C_VEL
LIN {X 0,Y 228.584,Z 1164.266,A -85,B 0,C 180,E1 8615.477,E2 8615.477} C_VEL
LIN {X 0,Y 216.325,Z 1180.294,A -85,B 0,C 180,E1 8612.548,E2 8612.548} C_VEL
LIN {X 0,Y 204.135,Z 1195.015,A -85,B 0,C 180,E1 8608.995,E2 8608.995} C_VEL
LIN {X 0,Y 192.295,Z 1208.519,A -85,B 0,C 180,E1 8604.717,E2 8604.717} C_VEL
LIN {X 0,Y 181.206,Z 1220.858,A -85,B 0,C 180,E1 8599.59,E2 8599.59} C_VEL
LIN {X 0,Y 171.363,Z 1231.825,A -85,B 0,C 180,E1 8593.51,E2 8593.51} C_VEL
LIN {X 0,Y 163.316,Z 1241.398,A -85,B 0,C 180,E1 8586.43,E2 8586.43} C_VEL
LIN {X 0,Y 157.837,Z 1249.188,A -85,B 0,C 180,E1 8578.779,E2 8578.779} C_VEL
LIN {X 0,Y 154.966,Z 1255.184,A -85,B 0,C 180,E1 8570.785,E2 8570.785} C_VEL
LIN {X 0,Y 154.457,Z 1259.423,A -85,B 0,C 180,E1 8562.714,E2 8562.714} C_VEL
LIN {X 0,Y 155.186,Z 1261.471,A -85,B 0,C 180,E1 8556.66,E2 8556.66} C_VEL
LIN {X 0,Y 155.904,Z 1262.279,A -85,B 0,C 180,E1 8551.838,E2 8551.838} C_VEL
LIN {X 0,Y 155.904,Z 1262.276,A -85,B 0,C 180,E1 8548.162,E2 8548.162} C_VEL
LIN {X 0,Y 155.186,Z 1261.461,A -85,B 0,C 180,E1 8543.34,E2 8543.34} C_VEL
LIN {X 0,Y 154.459,Z 1259.406,A -85,B 0,C 180,E1 8537.286,E2 8537.286} C_VEL
LIN {X 0,Y 154.968,Z 1255.154,A -85,B 0,C 180,E1 8529.216,E2 8529.216} C_VEL
LIN {X 0,Y 157.644,Z 1249.466,A -85,B 0,C 180,E1 8521.597,E2 8521.597} C_VEL
LIN {X 0,Y 162.996,Z 1241.762,A -85,B 0,C 180,E1 8513.923,E2 8513.923} C_VEL
LIN {X 0,Y 170.922,Z 1232.275,A -85,B 0,C 180,E1 8506.811,E2 8506.811} C_VEL
LIN {X 0,Y 180.662,Z 1221.356,A -85,B 0,C 180,E1 8500.695,E2 8500.695} C_VEL
LIN {X 0,Y 191.671,Z 1209.117,A -85,B 0,C 180,E1 8495.536,E2 8495.536} C_VEL
LIN {X 0,Y 203.442,Z 1195.718,A -85,B 0,C 180,E1 8491.226,E2 8491.226} C_VEL
LIN {X 0,Y 215.672,Z 1180.938,A -85,B 0,C 180,E1 8487.619,E2 8487.619} C_VEL
LIN {X 0,Y 228.238,Z 1164.551,A -85,B 0,C 180,E1 8484.593,E2 8484.593} C_VEL
LIN {X 0,Y 240.634,Z 1146.814,A -85,B 0,C 180,E1 8482.096,E2 8482.096} C_VEL
LIN {X 0,Y 251.907,Z 1128.87,A -85,B 0,C 180,E1 8480.17,E2 8480.17} C_VEL
LIN {X 0,Y 262.223,Z 1110.169,A -85,B 0,C 180,E1 8478.648,E2 8478.648} C_VEL
LIN {X 0,Y 271.911,Z 1090.106,A -85,B 0,C 180,E1 8477.409,E2 8477.409} C_VEL
LIN {X 0,Y 280.433,Z 1069.344,A -85,B 0,C 180,E1 8476.451,E2 8476.451} C_VEL
LIN {X 0,Y 287.399,Z 1048.044,A -85,B 0,C 180,E1 8475.681,E2 8475.681} C_VEL
LIN {X 0,Y 293.129,Z 1025.194,A -85,B 0,C 180,E1 8475.016,E2 8475.016} C_VEL
LIN {X 0,Y 297.071,Z 1002.737,A -85,B 0,C 180,E1 8474.49,E2 8474.49} C_VEL
LIN {X 0,Y 309.334,Z 883.976,A -85,B 0,C 180,E1 8472.275,E2 8472.275} C_VEL
LIN {X 0,Y 307.407,Z 877.661,A -85,B 0,C 180,E1 8469.973,E2 8469.973} C_VEL
LIN {X 0,Y 305.67,Z 871.751,A -85,B 0,C 180,E1 8467.329,E2 8467.329} C_VEL
LIN {X 0,Y 304.389,Z 867.286,A -85,B 0,C 180,E1 8464.616,E2 8464.616} C_VEL
LIN {X 0,Y 303.97,Z 866.51,A -85,B 0,C 180,E1 8463.583,E2 8463.583} C_VEL
LIN {X 0,Y 303.069,Z 864.995,A -85,B 0,C 180,E1 8458.676,E2 8458.676} C_VEL
LIN {X 0,Y 304.257,Z 866.854,A -85,B 0,C 180,E1 8453.205,E2 8453.205} C_VEL
LIN {X 0,Y 306.349,Z 871.523,A -85,B 0,C 180,E1 8449.373,E2 8449.373} C_VEL
LIN {X 0,Y 308.5,Z 876.041,A -85,B 0,C 180,E1 8446.696,E2 8446.696} C_VEL
LIN {X 0,Y 309.383,Z 878.044,A -85,B 0,C 180,E1 8445.747,E2 8445.747} C_VEL
LIN {X 0,Y 301,Z 960.602,A -85,B 0,C 180,E1 8444.176,E2 8444.176} C_VEL
LIN {X 0,Y 298.155,Z 983.742,A -85,B 0,C 180,E1 8443.529,E2 8443.529} C_VEL
LIN {X 0,Y 293.927,Z 1005.735,A -85,B 0,C 180,E1 8442.706,E2 8442.706} C_VEL
LIN {X 0,Y 288.522,Z 1026.306,A -85,B 0,C 180,E1 8441.714,E2 8441.714} C_VEL
LIN {X 0,Y 281.744,Z 1046.172,A -85,B 0,C 180,E1 8440.513,E2 8440.513} C_VEL
LIN {X 0,Y 273.434,Z 1066.209,A -85,B 0,C 180,E1 8439,E2 8439} C_VEL
LIN {X 0,Y 264.458,Z 1084.478,A -85,B 0,C 180,E1 8437.292,E2 8437.292} C_VEL
LIN {X 0,Y 254.337,Z 1101.993,A -85,B 0,C 180,E1 8435.242,E2 8435.242} C_VEL
LIN {X 0,Y 243.352,Z 1118.589,A -85,B 0,C 180,E1 8432.811,E2 8432.811} C_VEL
LIN {X 0,Y 232.041,Z 1133.76,A -85,B 0,C 180,E1 8430.006,E2 8430.006} C_VEL
LIN {X 0,Y 220.202,Z 1147.893,A -85,B 0,C 180,E1 8426.663,E2 8426.663} C_VEL
LIN {X 0,Y 208.426,Z 1160.512,A -85,B 0,C 180,E1 8422.779,E2 8422.779} C_VEL
LIN {X 0,Y 196.404,Z 1172.29,A -85,B 0,C 180,E1 8418.008,E2 8418.008} C_VEL
LIN {X 0,Y 185.711,Z 1182.033,A -85,B 0,C 180,E1 8412.715,E2 8412.715} C_VEL
LIN {X 0,Y 176.094,Z 1190.246,A -85,B 0,C 180,E1 8406.596,E2 8406.596} C_VEL
LIN {X 0,Y 168.294,Z 1196.651,A -85,B 0,C 180,E1 8399.937,E2 8399.937} C_VEL
LIN {X 0,Y 162.263,Z 1201.665,A -85,B 0,C 180,E1 8392.436,E2 8392.436} C_VEL
LIN {X 0,Y 158.436,Z 1205.033,A -85,B 0,C 180,E1 8384.621,E2 8384.621} C_VEL
LIN {X 0,Y 156.535,Z 1206.764,A -85,B 0,C 180,E1 8376.97,E2 8376.97} C_VEL
LIN {X 0,Y 156.07,Z 1207.333,A -85,B 0,C 180,E1 8369.633,E2 8369.633} C_VEL
LIN {X 0,Y 156.638,Z 1206.681,A -85,B 0,C 180,E1 8362.297,E2 8362.297} C_VEL
LIN {X 0,Y 158.799,Z 1204.691,A -85,B 0,C 180,E1 8354.292,E2 8354.292} C_VEL
LIN {X 0,Y 162.932,Z 1201.206,A -85,B 0,C 180,E1 8346.492,E2 8346.492} C_VEL
LIN {X 0,Y 169.223,Z 1195.964,A -85,B 0,C 180,E1 8339.068,E2 8339.068} C_VEL
LIN {X 0,Y 177.699,Z 1188.944,A -85,B 0,C 180,E1 8332.172,E2 8332.172} C_VEL
LIN {X 0,Y 187.137,Z 1180.882,A -85,B 0,C 180,E1 8326.432,E2 8326.432} C_VEL
LIN {X 0,Y 198.031,Z 1170.922,A -85,B 0,C 180,E1 8321.212,E2 8321.212} C_VEL
LIN {X 0,Y 209.587,Z 1159.468,A -85,B 0,C 180,E1 8316.732,E2 8316.732} C_VEL
LIN {X 0,Y 222.023,Z 1145.949,A -85,B 0,C 180,E1 8312.712,E2 8312.712} C_VEL
LIN {X 0,Y 233.836,Z 1131.723,A -85,B 0,C 180,E1 8309.455,E2 8309.455} C_VEL
LIN {X 0,Y 245.118,Z 1116.352,A -85,B 0,C 180,E1 8306.71,E2 8306.71} C_VEL
LIN {X 0,Y 255.773,Z 1099.914,A -85,B 0,C 180,E1 8304.383,E2 8304.383} C_VEL
LIN {X 0,Y 265.539,Z 1082.767,A -85,B 0,C 180,E1 8302.426,E2 8302.426} C_VEL
LIN {X 0,Y 274.287,Z 1064.776,A -85,B 0,C 180,E1 8300.774,E2 8300.774} C_VEL
LIN {X 0,Y 282.341,Z 1045.087,A -85,B 0,C 180,E1 8299.312,E2 8299.312} C_VEL
LIN {X 0,Y 288.894,Z 1025.666,A -85,B 0,C 180,E1 8298.149,E2 8298.149} C_VEL
LIN {X 0,Y 294.405,Z 1004.555,A -85,B 0,C 180,E1 8297.142,E2 8297.142} C_VEL
LIN {X 0,Y 298.465,Z 983.013,A -85,B 0,C 180,E1 8296.347,E2 8296.347} C_VEL
LIN {X 0,Y 301.418,Z 958.294,A -85,B 0,C 180,E1 8295.67,E2 8295.67} C_VEL
LIN {X 0,Y 309.553,Z 877.947,A -85,B 0,C 180,E1 8294.115,E2 8294.115} C_VEL
LIN {X 0,Y 307.221,Z 873.139,A -85,B 0,C 180,E1 8291.451,E2 8291.451} C_VEL
LIN {X 0,Y 305.817,Z 870.181,A -85,B 0,C 180,E1 8289.409,E2 8289.409} C_VEL
LIN {X 0,Y 304.284,Z 866.716,A -85,B 0,C 180,E1 8286.226,E2 8286.226} C_VEL
LIN {X 0,Y 303.298,Z 865.317,A -85,B 0,C 180,E1 8280.945,E2 8280.945} C_VEL
LIN {X 0,Y 304.463,Z 867.041,A -85,B 0,C 180,E1 8275.763,E2 8275.763} C_VEL
LIN {X 0,Y 305.431,Z 870.372,A -85,B 0,C 180,E1 8273.516,E2 8273.516} C_VEL
LIN {X 0,Y 307.145,Z 876.161,A -85,B 0,C 180,E1 8270.68,E2 8270.68} C_VEL
LIN {X 0,Y 309.188,Z 883.019,A -85,B 0,C 180,E1 8268.103,E2 8268.103} C_VEL
LIN {X 0,Y 309.508,Z 884.325,A -85,B 0,C 180,E1 8267.724,E2 8267.724} C_VEL
LIN {X 0,Y 304.735,Z 931.004,A -85,B 0,C 180,E1 8266.872,E2 8266.872} C_VEL
LIN {X 0,Y 303.702,Z 938.7,A -85,B 0,C 180,E1 8266.915,E2 8266.915} C_VEL
LIN {X 0,Y 300.09,Z 959.238,A -85,B 0,C 180,E1 8267.692,E2 8267.692} C_VEL
LIN {X 0,Y 299.234,Z 965.841,A -85,B 0,C 180,E1 8267.71,E2 8267.71} C_VEL
LIN {X 0,Y 294.821,Z 1004.944,A -85,B 0,C 180,E1 8266.971,E2 8266.971} C_VEL
LIN {X 0,Y 290.544,Z 1027.414,A -85,B 0,C 180,E1 8266.446,E2 8266.446} C_VEL
LIN {X 0,Y 284.639,Z 1049.441,A -85,B 0,C 180,E1 8265.808,E2 8265.808} C_VEL
LIN {X 0,Y 276.88,Z 1071.803,A -85,B 0,C 180,E1 8265.007,E2 8265.007} C_VEL
LIN {X 0,Y 268.24,Z 1092.101,A -85,B 0,C 180,E1 8264.083,E2 8264.083} C_VEL
LIN {X 0,Y 258.4,Z 1111.521,A -85,B 0,C 180,E1 8262.885,E2 8262.885} C_VEL
LIN {X 0,Y 247.035,Z 1131.115,A -85,B 0,C 180,E1 8261.275,E2 8261.275} C_VEL
LIN {X 0,Y 235.505,Z 1148.764,A -85,B 0,C 180,E1 8259.367,E2 8259.367} C_VEL
LIN {X 0,Y 223.314,Z 1165.37,A -85,B 0,C 180,E1 8256.995,E2 8256.995} C_VEL
LIN {X 0,Y 210.303,Z 1181.52,A -85,B 0,C 180,E1 8253.968,E2 8253.968} C_VEL
LIN {X 0,Y 197.799,Z 1195.975,A -85,B 0,C 180,E1 8250.391,E2 8250.391} C_VEL
LIN {X 0,Y 184.957,Z 1209.818,A -85,B 0,C 180,E1 8245.792,E2 8245.792} C_VEL
LIN {X 0,Y 173.031,Z 1222.241,A -85,B 0,C 180,E1 8240.221,E2 8240.221} C_VEL
LIN {X 0,Y 162.456,Z 1233.402,A -85,B 0,C 180,E1 8233.428,E2 8233.428} C_VEL
LIN {X 0,Y 154.6,Z 1242.383,A -85,B 0,C 180,E1 8226.052,E2 8226.052} C_VEL
LIN {X 0,Y 149.142,Z 1249.889,A -85,B 0,C 180,E1 8217.553,E2 8217.553} C_VEL
LIN {X 0,Y 146.674,Z 1255.554,A -85,B 0,C 180,E1 8208.642,E2 8208.642} C_VEL
LIN {X 0,Y 146.715,Z 1259.079,A -85,B 0,C 180,E1 8200.603,E2 8200.603} C_VEL
LIN {X 0,Y 147.747,Z 1260.68,A -85,B 0,C 180,E1 8193.88,E2 8193.88} C_VEL
LIN {X 0,Y 148.109,Z 1261.005,A -85,B 0,C 180,E1 8189.613,E2 8189.613} C_VEL
LIN {X 0,Y 147.537,Z 1260.526,A -85,B 0,C 180,E1 8184.946,E2 8184.946} C_VEL
LIN {X 0,Y 146.602,Z 1258.595,A -85,B 0,C 180,E1 8178.194,E2 8178.194} C_VEL
LIN {X 0,Y 146.786,Z 1255.085,A -85,B 0,C 180,E1 8170.503,E2 8170.503} C_VEL
LIN {X 0,Y 149.51,Z 1249.231,A -85,B 0,C 180,E1 8161.654,E2 8161.654} C_VEL
LIN {X 0,Y 154.919,Z 1241.924,A -85,B 0,C 180,E1 8153.576,E2 8153.576} C_VEL
LIN {X 0,Y 163.031,Z 1232.735,A -85,B 0,C 180,E1 8146.132,E2 8146.132} C_VEL
LIN {X 0,Y 173.028,Z 1222.161,A -85,B 0,C 180,E1 8139.778,E2 8139.778} C_VEL
LIN {X 0,Y 184.963,Z 1209.708,A -85,B 0,C 180,E1 8134.203,E2 8134.203} C_VEL
LIN {X 0,Y 197.793,Z 1195.86,A -85,B 0,C 180,E1 8129.606,E2 8129.606} C_VEL
LIN {X 0,Y 210.298,Z 1181.376,A -85,B 0,C 180,E1 8126.029,E2 8126.029} C_VEL
LIN {X 0,Y 224.051,Z 1164.209,A -85,B 0,C 180,E1 8122.845,E2 8122.845} C_VEL
LIN {X 0,Y 236.388,Z 1147.251,A -85,B 0,C 180,E1 8120.47,E2 8120.47} C_VEL
LIN {X 0,Y 248.013,Z 1129.292,A -85,B 0,C 180,E1 8118.571,E2 8118.571} C_VEL
LIN {X 0,Y 258.793,Z 1110.469,A -85,B 0,C 180,E1 8117.059,E2 8117.059} C_VEL
LIN {X 0,Y 268.234,Z 1091.733,A -85,B 0,C 180,E1 8115.913,E2 8115.913} C_VEL
LIN {X 0,Y 276.873,Z 1071.356,A -85,B 0,C 180,E1 8114.988,E2 8114.988} C_VEL
LIN {X 0,Y 284.402,Z 1049.604,A -85,B 0,C 180,E1 8114.208,E2 8114.208} C_VEL
LIN {X 0,Y 290.308,Z 1027.625,A -85,B 0,C 180,E1 8113.571,E2 8113.571} C_VEL
LIN {X 0,Y 294.583,Z 1005.176,A -85,B 0,C 180,E1 8113.044,E2 8113.044} C_VEL
LIN {X 0,Y 298.872,Z 967.361,A -85,B 0,C 180,E1 8112.328,E2 8112.328} C_VEL
LIN {X 0,Y 307.025,Z 888.795,A -85,B 0,C 180,E1 8110.887,E2 8110.887} C_VEL
LIN {X 0,Y 304.802,Z 880.752,A -85,B 0,C 180,E1 8107.634,E2 8107.634} C_VEL
LIN {X 0,Y 303.39,Z 875.444,A -85,B 0,C 180,E1 8104.631,E2 8104.631} C_VEL
LIN {X 0,Y 302.994,Z 874.47,A -85,B 0,C 180,E1 8103.594,E2 8103.594} C_VEL
LIN {X 0,Y 302.094,Z 872.937,A -85,B 0,C 180,E1 8098.672,E2 8098.672} C_VEL
LIN {X 0,Y 303.194,Z 874.792,A -85,B 0,C 180,E1 8093.372,E2 8093.372} C_VEL
LIN {X 0,Y 305.099,Z 879.225,A -85,B 0,C 180,E1 8089.711,E2 8089.711} C_VEL
LIN {X 0,Y 307.086,Z 883.597,A -85,B 0,C 180,E1 8087.109,E2 8087.109} C_VEL
LIN {X 0,Y 298.952,Z 961.925,A -85,B 0,C 180,E1 8085.635,E2 8085.635} C_VEL
LIN {X 0,Y 296.04,Z 984.991,A -85,B 0,C 180,E1 8084.998,E2 8084.998} C_VEL
LIN {X 0,Y 291.733,Z 1006.925,A -85,B 0,C 180,E1 8084.193,E2 8084.193} C_VEL
LIN {X 0,Y 286.148,Z 1027.705,A -85,B 0,C 180,E1 8083.212,E2 8083.212} C_VEL
LIN {X 0,Y 279.132,Z 1047.79,A -85,B 0,C 180,E1 8082.023,E2 8082.023} C_VEL
LIN {X 0,Y 270.449,Z 1068.156,A -85,B 0,C 180,E1 8080.512,E2 8080.512} C_VEL
LIN {X 0,Y 261.109,Z 1086.579,A -85,B 0,C 180,E1 8078.812,E2 8078.812} C_VEL
LIN {X 0,Y 250.719,Z 1104.061,A -85,B 0,C 180,E1 8076.794,E2 8076.794} C_VEL
LIN {X 0,Y 239.46,Z 1120.515,A -85,B 0,C 180,E1 8074.406,E2 8074.406} C_VEL
LIN {X 0,Y 227.446,Z 1136.033,A -85,B 0,C 180,E1 8071.543,E2 8071.543} C_VEL
LIN {X 0,Y 215.249,Z 1150.086,A -85,B 0,C 180,E1 8068.215,E2 8068.215} C_VEL
LIN {X 0,Y 203.065,Z 1162.568,A -85,B 0,C 180,E1 8064.332,E2 8064.332} C_VEL
LIN {X 0,Y 191.172,Z 1173.695,A -85,B 0,C 180,E1 8059.781,E2 8059.781} C_VEL
LIN {X 0,Y 179.942,Z 1183.439,A -85,B 0,C 180,E1 8054.435,E2 8054.435} C_VEL
LIN {X 0,Y 169.765,Z 1191.653,A -85,B 0,C 180,E1 8048.199,E2 8048.199} C_VEL
LIN {X 0,Y 161.443,Z 1198.056,A -85,B 0,C 180,E1 8041.347,E2 8041.347} C_VEL
LIN {X 0,Y 154.96,Z 1203.058,A -85,B 0,C 180,E1 8033.58,E2 8033.58} C_VEL
LIN {X 0,Y 150.783,Z 1206.431,A -85,B 0,C 180,E1 8025.381,E2 8025.381} C_VEL
LIN {X 0,Y 148.704,Z 1208.157,A -85,B 0,C 180,E1 8017.34,E2 8017.34} C_VEL
LIN {X 0,Y 148.192,Z 1208.723,A -85,B 0,C 180,E1 8009.613,E2 8009.613} C_VEL
LIN {X 0,Y 148.755,Z 1208.129,A -85,B 0,C 180,E1 8002.275,E2 8002.275} C_VEL
LIN {X 0,Y 150.896,Z 1206.359,A -85,B 0,C 180,E1 7994.237,E2 7994.237} C_VEL
LIN {X 0,Y 155.164,Z 1202.961,A -85,B 0,C 180,E1 7986.049,E2 7986.049} C_VEL
LIN {X 0,Y 161.729,Z 1197.903,A -85,B 0,C 180,E1 7978.3,E2 7978.3} C_VEL
LIN {X 0,Y 170.572,Z 1191.078,A -85,B 0,C 180,E1 7971.157,E2 7971.157} C_VEL
LIN {X 0,Y 180.918,Z 1182.756,A -85,B 0,C 180,E1 7964.978,E2 7964.978} C_VEL
LIN {X 0,Y 192.275,Z 1172.852,A -85,B 0,C 180,E1 7959.682,E2 7959.682} C_VEL
LIN {X 0,Y 204.274,Z 1161.52,A -85,B 0,C 180,E1 7955.176,E2 7955.176} C_VEL
LIN {X 0,Y 216.543,Z 1148.808,A -85,B 0,C 180,E1 7951.33,E2 7951.33} C_VEL
LIN {X 0,Y 228.825,Z 1134.618,A -85,B 0,C 180,E1 7948.04,E2 7948.04} C_VEL
LIN {X 0,Y 240.55,Z 1119.27,A -85,B 0,C 180,E1 7945.278,E2 7945.278} C_VEL
LIN {X 0,Y 252.22,Z 1101.943,A -85,B 0,C 180,E1 7942.831,E2 7942.831} C_VEL
LIN {X 0,Y 262.23,Z 1084.932,A -85,B 0,C 180,E1 7940.911,E2 7940.911} C_VEL
LIN {X 0,Y 271.179,Z 1067.03,A -85,B 0,C 180,E1 7939.29,E2 7939.29} C_VEL
LIN {X 0,Y 279.42,Z 1047.566,A -85,B 0,C 180,E1 7937.86,E2 7937.86} C_VEL
LIN {X 0,Y 286.275,Z 1027.958,A -85,B 0,C 180,E1 7936.698,E2 7936.698} C_VEL
LIN {X 0,Y 292.002,Z 1006.652,A -85,B 0,C 180,E1 7935.695,E2 7935.695} C_VEL
LIN {X 0,Y 296.259,Z 984.903,A -85,B 0,C 180,E1 7934.899,E2 7934.899} C_VEL
LIN {X 0,Y 299.208,Z 961.417,A -85,B 0,C 180,E1 7934.254,E2 7934.254} C_VEL
LIN {X 0,Y 307.272,Z 883.734,A -85,B 0,C 180,E1 7932.784,E2 7932.784} C_VEL
LIN {X 0,Y 304.957,Z 878.473,A -85,B 0,C 180,E1 7929.626,E2 7929.626} C_VEL
LIN {X 0,Y 303.161,Z 874.535,A -85,B 0,C 180,E1 7925.869,E2 7925.869} C_VEL
LIN {X 0,Y 302.323,Z 873.259,A -85,B 0,C 180,E1 7920.948,E2 7920.948} C_VEL
LIN {X 0,Y 303.399,Z 874.965,A -85,B 0,C 180,E1 7915.937,E2 7915.937} C_VEL
LIN {X 0,Y 304.414,Z 878.708,A -85,B 0,C 180,E1 7913.494,E2 7913.494} C_VEL
LIN {X 0,Y 305.987,Z 884.593,A -85,B 0,C 180,E1 7910.787,E2 7910.787} C_VEL
LIN {X 0,Y 307.23,Z 889.128,A -85,B 0,C 180,E1 7909.091,E2 7909.091} C_VEL
LIN {X 0,Y 299.234,Z 965.841,A -85,B 0,C 180,E1 7907.71,E2 7907.71} C_VEL
LIN {X 0,Y 298.212,Z 973.538,A -85,B 0,C 180,E1 7907.759,E2 7907.759} C_VEL
LIN {X 0,Y 294.535,Z 994.051,A -85,B 0,C 180,E1 7908.573,E2 7908.573} C_VEL
LIN {X 0,Y 293.537,Z 1000.636,A -85,B 0,C 180,E1 7908.574,E2 7908.574} C_VEL
LIN {X 0,Y 289.412,Z 1022.938,A -85,B 0,C 180,E1 7908.084,E2 7908.084} C_VEL
LIN {X 0,Y 283.453,Z 1045.767,A -85,B 0,C 180,E1 7907.47,E2 7907.47} C_VEL
LIN {X 0,Y 276.285,Z 1066.935,A -85,B 0,C 180,E1 7906.771,E2 7906.771} C_VEL
LIN {X 0,Y 267.502,Z 1087.624,A -85,B 0,C 180,E1 7905.911,E2 7905.911} C_VEL
LIN {X 0,Y 257.467,Z 1107.588,A -85,B 0,C 180,E1 7904.797,E2 7904.797} C_VEL
LIN {X 0,Y 246.726,Z 1126.214,A -85,B 0,C 180,E1 7903.413,E2 7903.413} C_VEL
LIN {X 0,Y 234.921,Z 1144.12,A -85,B 0,C 180,E1 7901.639,E2 7901.639} C_VEL
LIN {X 0,Y 222.199,Z 1161.338,A -85,B 0,C 180,E1 7899.38,E2 7899.38} C_VEL
LIN {X 0,Y 209.155,Z 1177.353,A -85,B 0,C 180,E1 7896.609,E2 7896.609} C_VEL
LIN {X 0,Y 196.017,Z 1192.057,A -85,B 0,C 180,E1 7893.205,E2 7893.205} C_VEL
LIN {X 0,Y 183.076,Z 1205.548,A -85,B 0,C 180,E1 7889.028,E2 7889.028} C_VEL
LIN {X 0,Y 170.744,Z 1217.881,A -85,B 0,C 180,E1 7883.909,E2 7883.909} C_VEL
LIN {X 0,Y 159.015,Z 1229.362,A -85,B 0,C 180,E1 7877.362,E2 7877.362} C_VEL
LIN {X 0,Y 149.693,Z 1238.836,A -85,B 0,C 180,E1 7869.881,E2 7869.881} C_VEL
LIN {X 0,Y 142.64,Z 1247.165,A -85,B 0,C 180,E1 7860.776,E2 7860.776} C_VEL
LIN {X 0,Y 139.247,Z 1253.009,A -85,B 0,C 180,E1 7851.924,E2 7851.924} C_VEL
LIN {X 0,Y 138.574,Z 1256.856,A -85,B 0,C 180,E1 7843.349,E2 7843.349} C_VEL
LIN {X 0,Y 139.435,Z 1258.938,A -85,B 0,C 180,E1 7836.175,E2 7836.175} C_VEL
LIN {X 0,Y 140.181,Z 1259.558,A -85,B 0,C 180,E1 7831.226,E2 7831.226} C_VEL
LIN {X 0,Y 140.013,Z 1259.409,A -85,B 0,C 180,E1 7827.135,E2 7827.135} C_VEL
LIN {X 0,Y 138.991,Z 1258.206,A -85,B 0,C 180,E1 7820.894,E2 7820.894} C_VEL
LIN {X 0,Y 138.655,Z 1254.993,A -85,B 0,C 180,E1 7812.148,E2 7812.148} C_VEL
LIN {X 0,Y 140.675,Z 1250.131,A -85,B 0,C 180,E1 7803.4,E2 7803.4} C_VEL
LIN {X 0,Y 145.591,Z 1243.403,A -85,B 0,C 180,E1 7794.77,E2 7794.77} C_VEL
LIN {X 0,Y 153.376,Z 1234.965,A -85,B 0,C 180,E1 7786.806,E2 7786.806} C_VEL
LIN {X 0,Y 163.77,Z 1224.619,A -85,B 0,C 180,E1 7779.714,E2 7779.714} C_VEL
LIN {X 0,Y 175.748,Z 1212.797,A -85,B 0,C 180,E1 7773.84,E2 7773.84} C_VEL
LIN {X 0,Y 189.41,Z 1198.923,A -85,B 0,C 180,E1 7768.806,E2 7768.806} C_VEL
LIN {X 0,Y 202.858,Z 1184.399,A -85,B 0,C 180,E1 7764.922,E2 7764.922} C_VEL
LIN {X 0,Y 216.412,Z 1168.468,A -85,B 0,C 180,E1 7761.779,E2 7761.779} C_VEL
LIN {X 0,Y 229.344,Z 1151.662,A -85,B 0,C 180,E1 7759.294,E2 7759.294} C_VEL
LIN {X 0,Y 241.874,Z 1133.555,A -85,B 0,C 180,E1 7757.277,E2 7757.277} C_VEL
LIN {X 0,Y 252.958,Z 1115.442,A -85,B 0,C 180,E1 7755.752,E2 7755.752} C_VEL
LIN {X 0,Y 263.367,Z 1095.836,A -85,B 0,C 180,E1 7754.519,E2 7754.519} C_VEL
LIN {X 0,Y 273.034,Z 1074.51,A -85,B 0,C 180,E1 7753.533,E2 7753.533} C_VEL
LIN {X 0,Y 280.905,Z 1053.412,A -85,B 0,C 180,E1 7752.774,E2 7752.774} C_VEL
LIN {X 0,Y 287.273,Z 1031.262,A -85,B 0,C 180,E1 7752.135,E2 7752.135} C_VEL
LIN {X 0,Y 292.011,Z 1008.662,A -85,B 0,C 180,E1 7751.602,E2 7751.602} C_VEL
LIN {X 0,Y 295.353,Z 983.84,A -85,B 0,C 180,E1 7751.122,E2 7751.122} C_VEL
LIN {X 0,Y 304.892,Z 893.756,A -85,B 0,C 180,E1 7749.489,E2 7749.489} C_VEL
LIN {X 0,Y 303.167,Z 887.022,A -85,B 0,C 180,E1 7746.533,E2 7746.533} C_VEL
LIN {X 0,Y 302.093,Z 882.533,A -85,B 0,C 180,E1 7743.795,E2 7743.795} C_VEL
LIN {X 0,Y 301.119,Z 880.879,A -85,B 0,C 180,E1 7738.668,E2 7738.668} C_VEL
LIN {X 0,Y 302.104,Z 882.607,A -85,B 0,C 180,E1 7733.634,E2 7733.634} C_VEL
LIN {X 0,Y 303.86,Z 886.927,A -85,B 0,C 180,E1 7730.052,E2 7730.052} C_VEL
LIN {X 0,Y 304.941,Z 889.464,A -85,B 0,C 180,E1 7728.477,E2 7728.477} C_VEL
LIN {X 0,Y 297.167,Z 962.583,A -85,B 0,C 180,E1 7727.129,E2 7727.129} C_VEL
LIN {X 0,Y 294.149,Z 986.081,A -85,B 0,C 180,E1 7726.493,E2 7726.493} C_VEL
LIN {X 0,Y 289.819,Z 1007.797,A -85,B 0,C 180,E1 7725.715,E2 7725.715} C_VEL
LIN {X 0,Y 284.184,Z 1028.385,A -85,B 0,C 180,E1 7724.77,E2 7724.77} C_VEL
LIN {X 0,Y 277.182,Z 1048.202,A -85,B 0,C 180,E1 7723.636,E2 7723.636} C_VEL
LIN {X 0,Y 268.741,Z 1067.865,A -85,B 0,C 180,E1 7722.236,E2 7722.236} C_VEL
LIN {X 0,Y 259.194,Z 1086.547,A -85,B 0,C 180,E1 7720.587,E2 7720.587} C_VEL
LIN {X 0,Y 248.544,Z 1104.149,A -85,B 0,C 180,E1 7718.633,E2 7718.633} C_VEL
LIN {X 0,Y 236.94,Z 1120.859,A -85,B 0,C 180,E1 7716.303,E2 7716.303} C_VEL
LIN {X 0,Y 224.996,Z 1136.042,A -85,B 0,C 180,E1 7713.615,E2 7713.615} C_VEL
LIN {X 0,Y 212.313,Z 1150.245,A -85,B 0,C 180,E1 7710.364,E2 7710.364} C_VEL
LIN {X 0,Y 199.724,Z 1162.837,A -85,B 0,C 180,E1 7706.586,E2 7706.586} C_VEL
LIN {X 0,Y 187.371,Z 1174.063,A -85,B 0,C 180,E1 7702.144,E2 7702.144} C_VEL
LIN {X 0,Y 175.466,Z 1183.969,A -85,B 0,C 180,E1 7696.833,E2 7696.833} C_VEL
LIN {X 0,Y 164.994,Z 1191.967,A -85,B 0,C 180,E1 7690.878,E2 7690.878} C_VEL
LIN {X 0,Y 155.454,Z 1198.929,A -85,B 0,C 180,E1 7683.581,E2 7683.581} C_VEL
LIN {X 0,Y 148.531,Z 1203.93,A -85,B 0,C 180,E1 7675.947,E2 7675.947} C_VEL
LIN {X 0,Y 143.623,Z 1207.426,A -85,B 0,C 180,E1 7667.418,E2 7667.418} C_VEL
LIN {X 0,Y 141.015,Z 1209.441,A -85,B 0,C 180,E1 7658.563,E2 7658.563} C_VEL
LIN {X 0,Y 140.314,Z 1210.084,A -85,B 0,C 180,E1 7650.817,E2 7650.817} C_VEL
LIN {X 0,Y 140.81,Z 1209.632,A -85,B 0,C 180,E1 7642.657,E2 7642.657} C_VEL
LIN {X 0,Y 142.839,Z 1208.092,A -85,B 0,C 180,E1 7634.574,E2 7634.574} C_VEL
LIN {X 0,Y 147.151,Z 1204.893,A -85,B 0,C 180,E1 7625.941,E2 7625.941} C_VEL
LIN {X 0,Y 154.268,Z 1199.841,A -85,B 0,C 180,E1 7617.457,E2 7617.457} C_VEL
LIN {X 0,Y 163.042,Z 1193.576,A -85,B 0,C 180,E1 7610.375,E2 7610.375} C_VEL
LIN {X 0,Y 173.699,Z 1185.434,A -85,B 0,C 180,E1 7603.986,E2 7603.986} C_VEL
LIN {X 0,Y 185.416,Z 1175.837,A -85,B 0,C 180,E1 7598.566,E2 7598.566} C_VEL
LIN {X 0,Y 197.764,Z 1164.875,A -85,B 0,C 180,E1 7593.991,E2 7593.991} C_VEL
LIN {X 0,Y 210.355,Z 1152.502,A -85,B 0,C 180,E1 7590.111,E2 7590.111} C_VEL
LIN {X 0,Y 222.926,Z 1138.633,A -85,B 0,C 180,E1 7586.808,E2 7586.808} C_VEL
LIN {X 0,Y 235.663,Z 1122.827,A -85,B 0,C 180,E1 7583.896,E2 7583.896} C_VEL
LIN {X 0,Y 247.243,Z 1106.522,A -85,B 0,C 180,E1 7581.55,E2 7581.55} C_VEL
LIN {X 0,Y 257.859,Z 1089.176,A -85,B 0,C 180,E1 7579.574,E2 7579.574} C_VEL
LIN {X 0,Y 267.419,Z 1071.018,A -85,B 0,C 180,E1 7577.913,E2 7577.913} C_VEL
LIN {X 0,Y 275.84,Z 1052.232,A -85,B 0,C 180,E1 7576.52,E2 7576.52} C_VEL
LIN {X 0,Y 283.042,Z 1032.506,A -85,B 0,C 180,E1 7575.344,E2 7575.344} C_VEL
LIN {X 0,Y 289.141,Z 1011.335,A -85,B 0,C 180,E1 7574.335,E2 7574.335} C_VEL
LIN {X 0,Y 293.707,Z 990.111,A -85,B 0,C 180,E1 7573.539,E2 7573.539} C_VEL
LIN {X 0,Y 296.697,Z 969.06,A -85,B 0,C 180,E1 7572.934,E2 7572.934} C_VEL
LIN {X 0,Y 302.015,Z 918.576,A -85,B 0,C 180,E1 7571.925,E2 7571.925} C_VEL
LIN {X 0,Y 305.132,Z 889.423,A -85,B 0,C 180,E1 7571.391,E2 7571.391} C_VEL
LIN {X 0,Y 303.401,Z 885.599,A -85,B 0,C 180,E1 7568.72,E2 7568.72} C_VEL
LIN {X 0,Y 302.117,Z 882.427,A -85,B 0,C 180,E1 7565.698,E2 7565.698} C_VEL
LIN {X 0,Y 301.348,Z 881.201,A -85,B 0,C 180,E1 7560.951,E2 7560.951} C_VEL
LIN {X 0,Y 302.308,Z 882.769,A -85,B 0,C 180,E1 7556.208,E2 7556.208} C_VEL
LIN {X 0,Y 303.249,Z 886.629,A -85,B 0,C 180,E1 7553.754,E2 7553.754} C_VEL
LIN {X 0,Y 304.742,Z 892.649,A -85,B 0,C 180,E1 7551.034,E2 7551.034} C_VEL
LIN {X 0,Y 305.094,Z 894.25,A -85,B 0,C 180,E1 7550.473,E2 7550.473} C_VEL
LIN {X 0,Y 293.537,Z 1000.636,A -85,B 0,C 180,E1 7548.574,E2 7548.574} C_VEL
LIN {X 0,Y 292.173,Z 1008.273,A -85,B 0,C 180,E1 7548.6,E2 7548.6} C_VEL
LIN {X 0,Y 286.426,Z 1028.379,A -85,B 0,C 180,E1 7549.367,E2 7549.367} C_VEL
LIN {X 0,Y 284.562,Z 1034.79,A -85,B 0,C 180,E1 7549.339,E2 7549.339} C_VEL
LIN {X 0,Y 277.354,Z 1057.779,A -85,B 0,C 180,E1 7548.674,E2 7548.674} C_VEL
LIN {X 0,Y 269.382,Z 1078.023,A -85,B 0,C 180,E1 7547.958,E2 7547.958} C_VEL
LIN {X 0,Y 259.595,Z 1098.43,A -85,B 0,C 180,E1 7547.014,E2 7547.014} C_VEL
LIN {X 0,Y 248.584,Z 1118.061,A -85,B 0,C 180,E1 7545.772,E2 7545.772} C_VEL
LIN {X 0,Y 236.884,Z 1136.347,A -85,B 0,C 180,E1 7544.224,E2 7544.224} C_VEL
LIN {X 0,Y 224.143,Z 1153.89,A -85,B 0,C 180,E1 7542.242,E2 7542.242} C_VEL
LIN {X 0,Y 210.639,Z 1170.47,A -85,B 0,C 180,E1 7539.726,E2 7539.726} C_VEL
LIN {X 0,Y 196.298,Z 1186.446,A -85,B 0,C 180,E1 7536.465,E2 7536.465} C_VEL
LIN {X 0,Y 182.539,Z 1200.589,A -85,B 0,C 180,E1 7532.54,E2 7532.54} C_VEL
LIN {X 0,Y 169.179,Z 1213.299,A -85,B 0,C 180,E1 7527.684,E2 7527.684} C_VEL
LIN {X 0,Y 156.195,Z 1225.278,A -85,B 0,C 180,E1 7521.347,E2 7521.347} C_VEL
LIN {X 0,Y 145.491,Z 1235.283,A -85,B 0,C 180,E1 7513.954,E2 7513.954} C_VEL
LIN {X 0,Y 137.375,Z 1243.559,A -85,B 0,C 180,E1 7505.397,E2 7505.397} C_VEL
LIN {X 0,Y 132.394,Z 1250.002,A -85,B 0,C 180,E1 7495.977,E2 7495.977} C_VEL
LIN {X 0,Y 130.618,Z 1254.766,A -85,B 0,C 180,E1 7485.996,E2 7485.996} C_VEL
LIN {X 0,Y 131.181,Z 1257.108,A -85,B 0,C 180,E1 7478.326,E2 7478.326} C_VEL
LIN {X 0,Y 132.206,Z 1258.095,A -85,B 0,C 180,E1 7472.167,E2 7472.167} C_VEL
LIN {X 0,Y 132.251,Z 1258.128,A -85,B 0,C 180,E1 7468.267,E2 7468.267} C_VEL
LIN {X 0,Y 131.317,Z 1257.306,A -85,B 0,C 180,E1 7462.563,E2 7462.563} C_VEL
LIN {X 0,Y 130.614,Z 1255.071,A -85,B 0,C 180,E1 7454.914,E2 7454.914} C_VEL
LIN {X 0,Y 132.097,Z 1250.491,A -85,B 0,C 180,E1 7444.922,E2 7444.922} C_VEL
LIN {X 0,Y 136.893,Z 1244.08,A -85,B 0,C 180,E1 7435.272,E2 7435.272} C_VEL
LIN {X 0,Y 145.044,Z 1235.641,A -85,B 0,C 180,E1 7426.423,E2 7426.423} C_VEL
LIN {X 0,Y 155.627,Z 1225.72,A -85,B 0,C 180,E1 7418.98,E2 7418.98} C_VEL
LIN {X 0,Y 168.09,Z 1214.239,A -85,B 0,C 180,E1 7412.771,E2 7412.771} C_VEL
LIN {X 0,Y 181.799,Z 1201.188,A -85,B 0,C 180,E1 7407.694,E2 7407.694} C_VEL
LIN {X 0,Y 195.502,Z 1187.133,A -85,B 0,C 180,E1 7403.733,E2 7403.733} C_VEL
LIN {X 0,Y 210.113,Z 1170.908,A -85,B 0,C 180,E1 7400.376,E2 7400.376} C_VEL
LIN {X 0,Y 223.704,Z 1154.256,A -85,B 0,C 180,E1 7397.827,E2 7397.827} C_VEL
LIN {X 0,Y 236.432,Z 1136.739,A -85,B 0,C 180,E1 7395.834,E2 7395.834} C_VEL
LIN {X 0,Y 248.123,Z 1118.525,A -85,B 0,C 180,E1 7394.278,E2 7394.278} C_VEL
LIN {X 0,Y 259.127,Z 1098.987,A -85,B 0,C 180,E1 7393.029,E2 7393.029} C_VEL
LIN {X 0,Y 268.908,Z 1078.627,A -85,B 0,C 180,E1 7392.078,E2 7392.078} C_VEL
LIN {X 0,Y 276.878,Z 1058.542,A -85,B 0,C 180,E1 7391.361,E2 7391.361} C_VEL
LIN {X 0,Y 283.902,Z 1036.511,A -85,B 0,C 180,E1 7390.715,E2 7390.715} C_VEL
LIN {X 0,Y 289.281,Z 1014.039,A -85,B 0,C 180,E1 7390.175,E2 7390.175} C_VEL
LIN {X 0,Y 292.848,Z 991.326,A -85,B 0,C 180,E1 7389.728,E2 7389.728} C_VEL
LIN {X 0,Y 302.933,Z 899.056,A -85,B 0,C 180,E1 7388.111,E2 7388.111} C_VEL
LIN {X 0,Y 301.686,Z 893.438,A -85,B 0,C 180,E1 7385.515,E2 7385.515} C_VEL
LIN {X 0,Y 300.969,Z 890.317,A -85,B 0,C 180,E1 7383.428,E2 7383.428} C_VEL
LIN {X 0,Y 300.145,Z 888.839,A -85,B 0,C 180,E1 7378.473,E2 7378.473} C_VEL
LIN {X 0,Y 301.077,Z 890.66,A -85,B 0,C 180,E1 7373.708,E2 7373.708} C_VEL
LIN {X 0,Y 302.632,Z 894.628,A -85,B 0,C 180,E1 7370.395,E2 7370.395} C_VEL
LIN {X 0,Y 302.924,Z 895.716,A -85,B 0,C 180,E1 7369.862,E2 7369.862} C_VEL
LIN {X 0,Y 295.521,Z 963.877,A -85,B 0,C 180,E1 7368.625,E2 7368.625} C_VEL
LIN {X 0,Y 292.407,Z 987.489,A -85,B 0,C 180,E1 7367.996,E2 7367.996} C_VEL
LIN {X 0,Y 287.967,Z 1009.23,A -85,B 0,C 180,E1 7367.233,E2 7367.233} C_VEL
LIN {X 0,Y 282.217,Z 1029.785,A -85,B 0,C 180,E1 7366.313,E2 7366.313} C_VEL
LIN {X 0,Y 275.067,Z 1049.599,A -85,B 0,C 180,E1 7365.21,E2 7365.21} C_VEL
LIN {X 0,Y 266.466,Z 1069.213,A -85,B 0,C 180,E1 7363.854,E2 7363.854} C_VEL
LIN {X 0,Y 256.681,Z 1087.944,A -85,B 0,C 180,E1 7362.247,E2 7362.247} C_VEL
LIN {X 0,Y 245.778,Z 1105.546,A -85,B 0,C 180,E1 7360.347,E2 7360.347} C_VEL
LIN {X 0,Y 233.875,Z 1122.257,A -85,B 0,C 180,E1 7358.077,E2 7358.077} C_VEL
LIN {X 0,Y 221.813,Z 1137.197,A -85,B 0,C 180,E1 7355.499,E2 7355.499} C_VEL
LIN {X 0,Y 208.684,Z 1151.458,A -85,B 0,C 180,E1 7352.305,E2 7352.305} C_VEL
LIN {X 0,Y 195.604,Z 1164.111,A -85,B 0,C 180,E1 7348.574,E2 7348.574} C_VEL
LIN {X 0,Y 182.621,Z 1175.451,A -85,B 0,C 180,E1 7344.123,E2 7344.123} C_VEL
LIN {X 0,Y 170.119,Z 1185.376,A -85,B 0,C 180,E1 7338.789,E2 7338.789} C_VEL
LIN {X 0,Y 158.549,Z 1193.739,A -85,B 0,C 180,E1 7332.435,E2 7332.435} C_VEL
LIN {X 0,Y 148.477,Z 1200.602,A -85,B 0,C 180,E1 7324.916,E2 7324.916} C_VEL
LIN {X 0,Y 140.824,Z 1205.688,A -85,B 0,C 180,E1 7316.57,E2 7316.57} C_VEL
LIN {X 0,Y 135.729,Z 1209.095,A -85,B 0,C 180,E1 7307.579,E2 7307.579} C_VEL
LIN {X 0,Y 133.135,Z 1210.889,A -85,B 0,C 180,E1 7298.638,E2 7298.638} C_VEL
LIN {X 0,Y 132.44,Z 1211.514,A -85,B 0,C 180,E1 7290,E2 7290} C_VEL
LIN {X 0,Y 133.125,Z 1210.915,A -85,B 0,C 180,E1 7281.361,E2 7281.361} C_VEL
LIN {X 0,Y 135.701,Z 1209.157,A -85,B 0,C 180,E1 7272.417,E2 7272.417} C_VEL
LIN {X 0,Y 140.778,Z 1205.766,A -85,B 0,C 180,E1 7263.421,E2 7263.421} C_VEL
LIN {X 0,Y 148.41,Z 1200.713,A -85,B 0,C 180,E1 7255.065,E2 7255.065} C_VEL
LIN {X 0,Y 158.469,Z 1193.889,A -85,B 0,C 180,E1 7247.538,E2 7247.538} C_VEL
LIN {X 0,Y 170.034,Z 1185.563,A -85,B 0,C 180,E1 7241.178,E2 7241.178} C_VEL
LIN {X 0,Y 182.528,Z 1175.656,A -85,B 0,C 180,E1 7235.836,E2 7235.836} C_VEL
LIN {X 0,Y 195.551,Z 1164.32,A -85,B 0,C 180,E1 7231.367,E2 7231.367} C_VEL
LIN {X 0,Y 208.734,Z 1151.602,A -85,B 0,C 180,E1 7227.608,E2 7227.608} C_VEL
LIN {X 0,Y 221.819,Z 1137.407,A -85,B 0,C 180,E1 7224.426,E2 7224.426} C_VEL
LIN {X 0,Y 234.022,Z 1122.331,A -85,B 0,C 180,E1 7221.821,E2 7221.821} C_VEL
LIN {X 0,Y 246.107,Z 1105.359,A -85,B 0,C 180,E1 7219.522,E2 7219.522} C_VEL
LIN {X 0,Y 257.022,Z 1087.707,A -85,B 0,C 180,E1 7217.624,E2 7217.624} C_VEL
LIN {X 0,Y 266.388,Z 1069.801,A -85,B 0,C 180,E1 7216.088,E2 7216.088} C_VEL
LIN {X 0,Y 274.996,Z 1050.333,A -85,B 0,C 180,E1 7214.733,E2 7214.733} C_VEL
LIN {X 0,Y 282.15,Z 1030.722,A -85,B 0,C 180,E1 7213.631,E2 7213.631} C_VEL
LIN {X 0,Y 288.135,Z 1009.419,A -85,B 0,C 180,E1 7212.675,E2 7212.675} C_VEL
LIN {X 0,Y 292.595,Z 987.677,A -85,B 0,C 180,E1 7211.912,E2 7211.912} C_VEL
LIN {X 0,Y 295.7,Z 964.28,A -85,B 0,C 180,E1 7211.287,E2 7211.287} C_VEL
LIN {X 0,Y 302.734,Z 899.478,A -85,B 0,C 180,E1 7210.104,E2 7210.104} C_VEL
LIN {X 0,Y 303.148,Z 895.593,A -85,B 0,C 180,E1 7210.02,E2 7210.02} C_VEL
LIN {X 0,Y 302.111,Z 893.113,A -85,B 0,C 180,E1 7208.182,E2 7208.182} C_VEL
LIN {X 0,Y 301.076,Z 890.318,A -85,B 0,C 180,E1 7205.527,E2 7205.527} C_VEL
LIN {X 0,Y 300.373,Z 889.143,A -85,B 0,C 180,E1 7200.954,E2 7200.954} C_VEL
LIN {X 0,Y 301.252,Z 890.689,A -85,B 0,C 180,E1 7196.385,E2 7196.385} C_VEL
LIN {X 0,Y 302.26,Z 895.272,A -85,B 0,C 180,E1 7193.638,E2 7193.638} C_VEL
LIN {X 0,Y 303.132,Z 899.436,A -85,B 0,C 180,E1 7191.872,E2 7191.872} C_VEL
LIN {X 0,Y 291.936,Z 1000.007,A -85,B 0,C 180,E1 7190.121,E2 7190.121} C_VEL
LIN {X 0,Y 287.609,Z 1022.599,A -85,B 0,C 180,E1 7189.639,E2 7189.639} C_VEL
LIN {X 0,Y 284.562,Z 1034.79,A -85,B 0,C 180,E1 7189.339,E2 7189.339} C_VEL
LIN {X 0,Y 282.238,Z 1042.233,A -85,B 0,C 180,E1 7189.343,E2 7189.343} C_VEL
LIN {X 0,Y 274.603,Z 1060.583,A -85,B 0,C 180,E1 7190.001,E2 7190.001} C_VEL
LIN {X 0,Y 271.536,Z 1067.697,A -85,B 0,C 180,E1 7189.964,E2 7189.964} C_VEL
LIN {X 0,Y 262.601,Z 1087.815,A -85,B 0,C 180,E1 7189.207,E2 7189.207} C_VEL
LIN {X 0,Y 252.275,Z 1107.208,A -85,B 0,C 180,E1 7188.215,E2 7188.215} C_VEL
LIN {X 0,Y 240.254,Z 1126.773,A -85,B 0,C 180,E1 7186.856,E2 7186.856} C_VEL
LIN {X 0,Y 227.558,Z 1144.904,A -85,B 0,C 180,E1 7185.155,E2 7185.155} C_VEL
LIN {X 0,Y 214.285,Z 1161.607,A -85,B 0,C 180,E1 7183.039,E2 7183.039} C_VEL
LIN {X 0,Y 200.579,Z 1177.109,A -85,B 0,C 180,E1 7180.409,E2 7180.409} C_VEL
LIN {X 0,Y 186.646,Z 1191.538,A -85,B 0,C 180,E1 7177.128,E2 7177.128} C_VEL
LIN {X 0,Y 172.028,Z 1205.352,A -85,B 0,C 180,E1 7172.778,E2 7172.778} C_VEL
LIN {X 0,Y 158.027,Z 1217.775,A -85,B 0,C 180,E1 7167.297,E2 7167.297} C_VEL
LIN {X 0,Y 145.255,Z 1228.79,A -85,B 0,C 180,E1 7160.437,E2 7160.437} C_VEL
LIN {X 0,Y 134.969,Z 1237.922,A -85,B 0,C 180,E1 7152.385,E2 7152.385} C_VEL
LIN {X 0,Y 127.47,Z 1245.356,A -85,B 0,C 180,E1 7142.936,E2 7142.936} C_VEL
LIN {X 0,Y 123.393,Z 1251.147,A -85,B 0,C 180,E1 7132.385,E2 7132.385} C_VEL
LIN {X 0,Y 122.761,Z 1254.765,A -85,B 0,C 180,E1 7122.703,E2 7122.703} C_VEL
LIN {X 0,Y 123.881,Z 1256.457,A -85,B 0,C 180,E1 7114.629,E2 7114.629} C_VEL
LIN {X 0,Y 124.481,Z 1256.853,A -85,B 0,C 180,E1 7110,E2 7110} C_VEL
LIN {X 0,Y 123.88,Z 1256.454,A -85,B 0,C 180,E1 7105.371,E2 7105.371} C_VEL
LIN {X 0,Y 122.762,Z 1254.745,A -85,B 0,C 180,E1 7097.297,E2 7097.297} C_VEL
LIN {X 0,Y 123.394,Z 1251.119,A -85,B 0,C 180,E1 7087.615,E2 7087.615} C_VEL
LIN {X 0,Y 127.47,Z 1245.315,A -85,B 0,C 180,E1 7077.064,E2 7077.064} C_VEL
LIN {X 0,Y 134.968,Z 1237.868,A -85,B 0,C 180,E1 7067.614,E2 7067.614} C_VEL
LIN {X 0,Y 145.253,Z 1228.721,A -85,B 0,C 180,E1 7059.562,E2 7059.562} C_VEL
LIN {X 0,Y 158.024,Z 1217.686,A -85,B 0,C 180,E1 7052.701,E2 7052.701} C_VEL
LIN {X 0,Y 172.024,Z 1205.24,A -85,B 0,C 180,E1 7047.22,E2 7047.22} C_VEL
LIN {X 0,Y 186.641,Z 1191.41,A -85,B 0,C 180,E1 7042.869,E2 7042.869} C_VEL
LIN {X 0,Y 200.574,Z 1176.949,A -85,B 0,C 180,E1 7039.588,E2 7039.588} C_VEL
LIN {X 0,Y 215.151,Z 1160.344,A -85,B 0,C 180,E1 7036.803,E2 7036.803} C_VEL
LIN {X 0,Y 228.515,Z 1143.404,A -85,B 0,C 180,E1 7034.701,E2 7034.701} C_VEL
LIN {X 0,Y 241.165,Z 1125.121,A -85,B 0,C 180,E1 7033.026,E2 7033.026} C_VEL
LIN {X 0,Y 252.735,Z 1106.042,A -85,B 0,C 180,E1 7031.73,E2 7031.73} C_VEL
LIN {X 0,Y 262.597,Z 1087.411,A -85,B 0,C 180,E1 7030.788,E2 7030.788} C_VEL
LIN {X 0,Y 271.789,Z 1066.586,A -85,B 0,C 180,E1 7030.009,E2 7030.009} C_VEL
LIN {X 0,Y 279.427,Z 1045.283,A -85,B 0,C 180,E1 7029.365,E2 7029.365} C_VEL
LIN {X 0,Y 285.576,Z 1023.296,A -85,B 0,C 180,E1 7028.818,E2 7028.818} C_VEL
LIN {X 0,Y 290.062,Z 1000.816,A -85,B 0,C 180,E1 7028.354,E2 7028.354} C_VEL
LIN {X 0,Y 294.679,Z 962.58,A -85,B 0,C 180,E1 7027.688,E2 7027.688} C_VEL
LIN {X 0,Y 301.133,Z 904.259,A -85,B 0,C 180,E1 7026.673,E2 7026.673} C_VEL
LIN {X 0,Y 300.061,Z 898.756,A -85,B 0,C 180,E1 7023.725,E2 7023.725} C_VEL
LIN {X 0,Y 299.615,Z 897.834,A -85,B 0,C 180,E1 7022.295,E2 7022.295} C_VEL
LIN {X 0,Y 299.17,Z 896.783,A -85,B 0,C 180,E1 7018.468,E2 7018.468} C_VEL
LIN {X 0,Y 299.995,Z 898.472,A -85,B 0,C 180,E1 7013.973,E2 7013.973} C_VEL
LIN {X 0,Y 301.122,Z 901.658,A -85,B 0,C 180,E1 7011.269,E2 7011.269} C_VEL
LIN {X 0,Y 294.078,Z 965.171,A -85,B 0,C 180,E1 7010.136,E2 7010.136} C_VEL
LIN {X 0,Y 290.896,Z 988.739,A -85,B 0,C 180,E1 7009.521,E2 7009.521} C_VEL
LIN {X 0,Y 286.387,Z 1010.409,A -85,B 0,C 180,E1 7008.78,E2 7008.78} C_VEL
LIN {X 0,Y 280.677,Z 1030.466,A -85,B 0,C 180,E1 7007.91,E2 7007.91} C_VEL
LIN {X 0,Y 273.648,Z 1049.791,A -85,B 0,C 180,E1 7006.879,E2 7006.879} C_VEL
LIN {X 0,Y 265.262,Z 1068.872,A -85,B 0,C 180,E1 7005.623,E2 7005.623} C_VEL
LIN {X 0,Y 255.681,Z 1087.01,A -85,B 0,C 180,E1 7004.148,E2 7004.148} C_VEL
LIN {X 0,Y 245.237,Z 1103.944,A -85,B 0,C 180,E1 7002.439,E2 7002.439} C_VEL
LIN {X 0,Y 233.55,Z 1120.487,A -85,B 0,C 180,E1 7000.359,E2 7000.359} C_VEL
LIN {X 0,Y 221.178,Z 1135.658,A -85,B 0,C 180,E1 6997.925,E2 6997.925} C_VEL
LIN {X 0,Y 207.605,Z 1150.326,A -85,B 0,C 180,E1 6994.879,E2 6994.879} C_VEL
LIN {X 0,Y 193.85,Z 1163.519,A -85,B 0,C 180,E1 6991.26,E2 6991.26} C_VEL
LIN {X 0,Y 180.159,Z 1175.234,A -85,B 0,C 180,E1 6986.93,E2 6986.93} C_VEL
LIN {X 0,Y 167.487,Z 1184.901,A -85,B 0,C 180,E1 6981.997,E2 6981.997} C_VEL
LIN {X 0,Y 154.394,Z 1194.053,A -85,B 0,C 180,E1 6975.425,E2 6975.425} C_VEL
LIN {X 0,Y 143.784,Z 1200.955,A -85,B 0,C 180,E1 6968.205,E2 6968.205} C_VEL
LIN {X 0,Y 135.077,Z 1206.304,A -85,B 0,C 180,E1 6959.731,E2 6959.731} C_VEL
LIN {X 0,Y 128.992,Z 1209.957,A -85,B 0,C 180,E1 6950.414,E2 6950.414} C_VEL
LIN {X 0,Y 125.616,Z 1212.12,A -85,B 0,C 180,E1 6940.548,E2 6940.548} C_VEL
LIN {X 0,Y 124.576,Z 1212.825,A -85,B 0,C 180,E1 6931.84,E2 6931.84} C_VEL
LIN {X 0,Y 125.062,Z 1212.507,A -85,B 0,C 180,E1 6922.472,E2 6922.472} C_VEL
LIN {X 0,Y 127.292,Z 1211.071,A -85,B 0,C 180,E1 6913.575,E2 6913.575} C_VEL
LIN {X 0,Y 132.207,Z 1208.05,A -85,B 0,C 180,E1 6903.984,E2 6903.984} C_VEL
LIN {X 0,Y 139.459,Z 1203.718,A -85,B 0,C 180,E1 6895.502,E2 6895.502} C_VEL
LIN {X 0,Y 149.037,Z 1197.677,A -85,B 0,C 180,E1 6887.867,E2 6887.867} C_VEL
LIN {X 0,Y 160.623,Z 1189.909,A -85,B 0,C 180,E1 6881.133,E2 6881.133} C_VEL
LIN {X 0,Y 173.259,Z 1180.752,A -85,B 0,C 180,E1 6875.544,E2 6875.544} C_VEL
LIN {X 0,Y 186.436,Z 1170.165,A -85,B 0,C 180,E1 6870.901,E2 6870.901} C_VEL
LIN {X 0,Y 199.786,Z 1158.182,A -85,B 0,C 180,E1 6867.026,E2 6867.026} C_VEL
LIN {X 0,Y 213.05,Z 1144.915,A -85,B 0,C 180,E1 6863.777,E2 6863.777} C_VEL
LIN {X 0,Y 226.003,Z 1130.243,A -85,B 0,C 180,E1 6861.02,E2 6861.02} C_VEL
LIN {X 0,Y 238.078,Z 1114.592,A -85,B 0,C 180,E1 6858.736,E2 6858.736} C_VEL
LIN {X 0,Y 249.951,Z 1096.957,A -85,B 0,C 180,E1 6856.702,E2 6856.702} C_VEL
LIN {X 0,Y 260.386,Z 1078.955,A -85,B 0,C 180,E1 6855.049,E2 6855.049} C_VEL
LIN {X 0,Y 269.576,Z 1059.977,A -85,B 0,C 180,E1 6853.657,E2 6853.657} C_VEL
LIN {X 0,Y 277.532,Z 1040.219,A -85,B 0,C 180,E1 6852.484,E2 6852.484} C_VEL
LIN {X 0,Y 284.164,Z 1019.797,A -85,B 0,C 180,E1 6851.508,E2 6851.508} C_VEL
LIN {X 0,Y 289.156,Z 999.198,A -85,B 0,C 180,E1 6850.723,E2 6850.723} C_VEL
LIN {X 0,Y 292.892,Z 977.061,A -85,B 0,C 180,E1 6850.062,E2 6850.062} C_VEL
LIN {X 0,Y 297.534,Z 935.662,A -85,B 0,C 180,E1 6849.189,E2 6849.189} C_VEL
LIN {X 0,Y 301.331,Z 901.587,A -85,B 0,C 180,E1 6848.588,E2 6848.588} C_VEL
LIN {X 0,Y 300.038,Z 898.21,A -85,B 0,C 180,E1 6845.354,E2 6845.354} C_VEL
LIN {X 0,Y 299.398,Z 897.085,A -85,B 0,C 180,E1 6840.957,E2 6840.957} C_VEL
LIN {X 0,Y 300.199,Z 898.607,A -85,B 0,C 180,E1 6836.563,E2 6836.563} C_VEL
LIN {X 0,Y 301.142,Z 903.36,A -85,B 0,C 180,E1 6833.806,E2 6833.806} C_VEL
LIN {X 0,Y 301.341,Z 904.724,A -85,B 0,C 180,E1 6833.287,E2 6833.287} C_VEL
LIN {X 0,Y 290.649,Z 998.636,A -85,B 0,C 180,E1 6831.696,E2 6831.696} C_VEL
LIN {X 0,Y 286.261,Z 1021.18,A -85,B 0,C 180,E1 6831.237,E2 6831.237} C_VEL
LIN {X 0,Y 280.323,Z 1043.108,A -85,B 0,C 180,E1 6830.703,E2 6830.703} C_VEL
LIN {X 0,Y 273.03,Z 1064.087,A -85,B 0,C 180,E1 6830.087,E2 6830.087} C_VEL
LIN {X 0,Y 271.536,Z 1067.697,A -85,B 0,C 180,E1 6829.964,E2 6829.964} C_VEL
LIN {X 0,Y 268.303,Z 1074.909,A -85,B 0,C 180,E1 6829.922,E2 6829.922} C_VEL
LIN {X 0,Y 258.567,Z 1092.18,A -85,B 0,C 180,E1 6830.505,E2 6830.505} C_VEL
LIN {X 0,Y 254.673,Z 1098.869,A -85,B 0,C 180,E1 6830.407,E2 6830.407} C_VEL
LIN {X 0,Y 243.196,Z 1118.204,A -85,B 0,C 180,E1 6829.288,E2 6829.288} C_VEL
LIN {X 0,Y 230.636,Z 1136.604,A -85,B 0,C 180,E1 6827.839,E2 6827.839} C_VEL
LIN {X 0,Y 217.399,Z 1153.764,A -85,B 0,C 180,E1 6826.024,E2 6826.024} C_VEL
LIN {X 0,Y 203.16,Z 1170.103,A -85,B 0,C 180,E1 6823.672,E2 6823.672} C_VEL
LIN {X 0,Y 188.545,Z 1185.146,A -85,B 0,C 180,E1 6820.719,E2 6820.719} C_VEL
LIN {X 0,Y 173.827,Z 1199.024,A -85,B 0,C 180,E1 6816.969,E2 6816.969} C_VEL
LIN {X 0,Y 159.333,Z 1211.591,A -85,B 0,C 180,E1 6812.225,E2 6812.225} C_VEL
LIN {X 0,Y 145.589,Z 1222.817,A -85,B 0,C 180,E1 6806.198,E2 6806.198} C_VEL
LIN {X 0,Y 133.317,Z 1232.717,A -85,B 0,C 180,E1 6798.587,E2 6798.587} C_VEL
LIN {X 0,Y 123.811,Z 1240.802,A -85,B 0,C 180,E1 6789.64,E2 6789.64} C_VEL
LIN {X 0,Y 117.393,Z 1247.318,A -85,B 0,C 180,E1 6779.043,E2 6779.043} C_VEL
LIN {X 0,Y 114.836,Z 1252.024,A -85,B 0,C 180,E1 6767.742,E2 6767.742} C_VEL
LIN {X 0,Y 115.32,Z 1254.467,A -85,B 0,C 180,E1 6758.476,E2 6758.476} C_VEL
LIN {X 0,Y 116.495,Z 1255.377,A -85,B 0,C 180,E1 6751.475,E2 6751.475} C_VEL
LIN {X 0,Y 116.361,Z 1255.293,A -85,B 0,C 180,E1 6747.538,E2 6747.538} C_VEL
LIN {X 0,Y 115.181,Z 1254.239,A -85,B 0,C 180,E1 6740.507,E2 6740.507} C_VEL
LIN {X 0,Y 114.958,Z 1251.507,A -85,B 0,C 180,E1 6730.701,E2 6730.701} C_VEL
LIN {X 0,Y 117.815,Z 1246.755,A -85,B 0,C 180,E1 6719.954,E2 6719.954} C_VEL
LIN {X 0,Y 124.58,Z 1240.028,A -85,B 0,C 180,E1 6709.453,E2 6709.453} C_VEL
LIN {X 0,Y 134.373,Z 1231.829,A -85,B 0,C 180,E1 6700.628,E2 6700.628} C_VEL
LIN {X 0,Y 146.23,Z 1222.215,A -85,B 0,C 180,E1 6693.472,E2 6693.472} C_VEL
LIN {X 0,Y 160.798,Z 1210.225,A -85,B 0,C 180,E1 6687.232,E2 6687.232} C_VEL
LIN {X 0,Y 175.415,Z 1197.497,A -85,B 0,C 180,E1 6682.577,E2 6682.577} C_VEL
LIN {X 0,Y 190.228,Z 1183.348,A -85,B 0,C 180,E1 6678.903,E2 6678.903} C_VEL
LIN {X 0,Y 205.353,Z 1167.477,A -85,B 0,C 180,E1 6675.931,E2 6675.931} C_VEL
LIN {X 0,Y 219.658,Z 1150.75,A -85,B 0,C 180,E1 6673.639,E2 6673.639} C_VEL
LIN {X 0,Y 232.945,Z 1133.197,A -85,B 0,C 180,E1 6671.874,E2 6671.874} C_VEL
LIN {X 0,Y 245.072,Z 1114.874,A -85,B 0,C 180,E1 6670.513,E2 6670.513} C_VEL
LIN {X 0,Y 256.64,Z 1094.773,A -85,B 0,C 180,E1 6669.417,E2 6669.417} C_VEL
LIN {X 0,Y 266.624,Z 1074.39,A -85,B 0,C 180,E1 6668.613,E2 6668.613} C_VEL
LIN {X 0,Y 275.104,Z 1053.056,A -85,B 0,C 180,E1 6667.961,E2 6667.961} C_VEL
LIN {X 0,Y 282.114,Z 1030.771,A -85,B 0,C 180,E1 6667.401,E2 6667.401} C_VEL
LIN {X 0,Y 287.363,Z 1008.429,A -85,B 0,C 180,E1 6666.931,E2 6666.931} C_VEL
LIN {X 0,Y 290.892,Z 985.859,A -85,B 0,C 180,E1 6666.527,E2 6666.527} C_VEL
LIN {X 0,Y 299.509,Z 909.828,A -85,B 0,C 180,E1 6665.267,E2 6665.267} C_VEL
LIN {X 0,Y 298.878,Z 906.092,A -85,B 0,C 180,E1 6663.068,E2 6663.068} C_VEL
LIN {X 0,Y 298.195,Z 904.727,A -85,B 0,C 180,E1 6658.463,E2 6658.463} C_VEL
LIN {X 0,Y 298.945,Z 906.401,A -85,B 0,C 180,E1 6654.145,E2 6654.145} C_VEL
LIN {X 0,Y 299.419,Z 908.328,A -85,B 0,C 180,E1 6652.682,E2 6652.682} C_VEL
LIN {X 0,Y 292.774,Z 967.09,A -85,B 0,C 180,E1 6651.647,E2 6651.647} C_VEL
LIN {X 0,Y 289.543,Z 990.273,A -85,B 0,C 180,E1 6651.052,E2 6651.052} C_VEL
LIN {X 0,Y 284.913,Z 1011.981,A -85,B 0,C 180,E1 6650.329,E2 6650.329} C_VEL
LIN {X 0,Y 278.966,Z 1032.403,A -85,B 0,C 180,E1 6649.467,E2 6649.467} C_VEL
LIN {X 0,Y 271.473,Z 1052.393,A -85,B 0,C 180,E1 6648.427,E2 6648.427} C_VEL
LIN {X 0,Y 262.521,Z 1072.005,A -85,B 0,C 180,E1 6647.16,E2 6647.16} C_VEL
LIN {X 0,Y 252.32,Z 1090.736,A -85,B 0,C 180,E1 6645.66,E2 6645.66} C_VEL
LIN {X 0,Y 241.362,Z 1107.702,A -85,B 0,C 180,E1 6643.955,E2 6643.955} C_VEL
LIN {X 0,Y 228.445,Z 1125.053,A -85,B 0,C 180,E1 6641.757,E2 6641.757} C_VEL
LIN {X 0,Y 215.834,Z 1139.886,A -85,B 0,C 180,E1 6639.349,E2 6639.349} C_VEL
LIN {X 0,Y 201.956,Z 1154.109,A -85,B 0,C 180,E1 6636.331,E2 6636.331} C_VEL
LIN {X 0,Y 187.856,Z 1166.88,A -85,B 0,C 180,E1 6632.726,E2 6632.726} C_VEL
LIN {X 0,Y 173.781,Z 1178.26,A -85,B 0,C 180,E1 6628.375,E2 6628.375} C_VEL
LIN {X 0,Y 160.077,Z 1188.189,A -85,B 0,C 180,E1 6623.08,E2 6623.08} C_VEL
LIN {X 0,Y 147.181,Z 1196.554,A -85,B 0,C 180,E1 6616.625,E2 6616.625} C_VEL
LIN {X 0,Y 135.724,Z 1203.414,A -85,B 0,C 180,E1 6608.768,E2 6608.768} C_VEL
LIN {X 0,Y 126.807,Z 1208.495,A -85,B 0,C 180,E1 6599.784,E2 6599.784} C_VEL
LIN {X 0,Y 120.705,Z 1211.895,A -85,B 0,C 180,E1 6589.853,E2 6589.853} C_VEL
LIN {X 0,Y 117.547,Z 1213.676,A -85,B 0,C 180,E1 6579.794,E2 6579.794} C_VEL
LIN {X 0,Y 116.683,Z 1214.294,A -85,B 0,C 180,E1 6570,E2 6570} C_VEL
LIN {X 0,Y 117.537,Z 1213.701,A -85,B 0,C 180,E1 6560.205,E2 6560.205} C_VEL
LIN {X 0,Y 120.677,Z 1211.955,A -85,B 0,C 180,E1 6550.142,E2 6550.142} C_VEL
LIN {X 0,Y 126.784,Z 1208.558,A -85,B 0,C 180,E1 6540.171,E2 6540.171} C_VEL
LIN {X 0,Y 135.656,Z 1203.522,A -85,B 0,C 180,E1 6531.209,E2 6531.209} C_VEL
LIN {X 0,Y 147.103,Z 1196.7,A -85,B 0,C 180,E1 6523.343,E2 6523.343} C_VEL
LIN {X 0,Y 159.346,Z 1188.811,A -85,B 0,C 180,E1 6517.168,E2 6517.168} C_VEL
LIN {X 0,Y 172.977,Z 1178.988,A -85,B 0,C 180,E1 6511.823,E2 6511.823} C_VEL
LIN {X 0,Y 187.517,Z 1167.337,A -85,B 0,C 180,E1 6507.295,E2 6507.295} C_VEL
LIN {X 0,Y 201.539,Z 1154.728,A -85,B 0,C 180,E1 6503.694,E2 6503.694} C_VEL
LIN {X 0,Y 215.465,Z 1140.499,A -85,B 0,C 180,E1 6500.652,E2 6500.652} C_VEL
LIN {X 0,Y 228.368,Z 1125.421,A -85,B 0,C 180,E1 6498.185,E2 6498.185} C_VEL
LIN {X 0,Y 240.856,Z 1108.776,A -85,B 0,C 180,E1 6496.056,E2 6496.056} C_VEL
LIN {X 0,Y 252.251,Z 1091.223,A -85,B 0,C 180,E1 6494.28,E2 6494.28} C_VEL
LIN {X 0,Y 262.01,Z 1073.44,A -85,B 0,C 180,E1 6492.842,E2 6492.842} C_VEL
LIN {X 0,Y 271.416,Z 1053.1,A -85,B 0,C 180,E1 6491.514,E2 6491.514} C_VEL
LIN {X 0,Y 278.857,Z 1033.486,A -85,B 0,C 180,E1 6490.483,E2 6490.483} C_VEL
LIN {X 0,Y 285.114,Z 1012.093,A -85,B 0,C 180,E1 6489.579,E2 6489.579} C_VEL
LIN {X 0,Y 289.749,Z 990.43,A -85,B 0,C 180,E1 6488.857,E2 6488.857} C_VEL
LIN {X 0,Y 293.003,Z 967.146,A -85,B 0,C 180,E1 6488.258,E2 6488.258} C_VEL
LIN {X 0,Y 299.656,Z 908.239,A -85,B 0,C 180,E1 6487.198,E2 6487.198} C_VEL
LIN {X 0,Y 298.944,Z 906.032,A -85,B 0,C 180,E1 6484.989,E2 6484.989} C_VEL
LIN {X 0,Y 298.426,Z 905.053,A -85,B 0,C 180,E1 6480.768,E2 6480.768} C_VEL
LIN {X 0,Y 299.149,Z 906.524,A -85,B 0,C 180,E1 6476.743,E2 6476.743} C_VEL
LIN {X 0,Y 299.718,Z 910.171,A -85,B 0,C 180,E1 6474.715,E2 6474.715} C_VEL
LIN {X 0,Y 289.564,Z 997.396,A -85,B 0,C 180,E1 6473.282,E2 6473.282} C_VEL
LIN {X 0,Y 285.075,Z 1020.04,A -85,B 0,C 180,E1 6472.842,E2 6472.842} C_VEL
LIN {X 0,Y 278.947,Z 1042.25,A -85,B 0,C 180,E1 6472.332,E2 6472.332} C_VEL
LIN {X 0,Y 271.751,Z 1062.662,A -85,B 0,C 180,E1 6471.772,E2 6471.772} C_VEL
LIN {X 0,Y 262.635,Z 1083.341,A -85,B 0,C 180,E1 6471.075,E2 6471.075} C_VEL
LIN {X 0,Y 254.673,Z 1098.869,A -85,B 0,C 180,E1 6470.407,E2 6470.407} C_VEL
LIN {X 0,Y 250.572,Z 1105.586,A -85,B 0,C 180,E1 6470.276,E2 6470.276} C_VEL
LIN {X 0,Y 238.771,Z 1121.832,A -85,B 0,C 180,E1 6470.641,E2 6470.641} C_VEL
LIN {X 0,Y 234.296,Z 1127.916,A -85,B 0,C 180,E1 6470.433,E2 6470.433} C_VEL
LIN {X 0,Y 221.104,Z 1145.467,A -85,B 0,C 180,E1 6468.893,E2 6468.893} C_VEL
LIN {X 0,Y 207.309,Z 1161.8,A -85,B 0,C 180,E1 6466.963,E2 6466.963} C_VEL
LIN {X 0,Y 192.96,Z 1176.865,A -85,B 0,C 180,E1 6464.528,E2 6464.528} C_VEL
LIN {X 0,Y 177.391,Z 1191.607,A -85,B 0,C 180,E1 6461.244,E2 6461.244} C_VEL
LIN {X 0,Y 161.815,Z 1205.053,A -85,B 0,C 180,E1 6457.021,E2 6457.021} C_VEL
LIN {X 0,Y 146.672,Z 1217.095,A -85,B 0,C 180,E1 6451.565,E2 6451.565} C_VEL
LIN {X 0,Y 133.232,Z 1227.206,A -85,B 0,C 180,E1 6444.883,E2 6444.883} C_VEL
LIN {X 0,Y 121.054,Z 1236.411,A -85,B 0,C 180,E1 6435.936,E2 6435.936} C_VEL
LIN {X 0,Y 112.641,Z 1243.431,A -85,B 0,C 180,E1 6425.862,E2 6425.862} C_VEL
LIN {X 0,Y 107.917,Z 1248.643,A -85,B 0,C 180,E1 6414.64,E2 6414.64} C_VEL
LIN {X 0,Y 106.913,Z 1252.248,A -85,B 0,C 180,E1 6402.97,E2 6402.97} C_VEL
LIN {X 0,Y 108.11,Z 1253.739,A -85,B 0,C 180,E1 6394.243,E2 6394.243} C_VEL
LIN {X 0,Y 108.717,Z 1254.072,A -85,B 0,C 180,E1 6390,E2 6390} C_VEL
LIN {X 0,Y 107.909,Z 1253.625,A -85,B 0,C 180,E1 6384.684,E2 6384.684} C_VEL
LIN {X 0,Y 106.84,Z 1251.619,A -85,B 0,C 180,E1 6374.558,E2 6374.558} C_VEL
LIN {X 0,Y 108.526,Z 1247.754,A -85,B 0,C 180,E1 6363.165,E2 6363.165} C_VEL
LIN {X 0,Y 114.335,Z 1241.824,A -85,B 0,C 180,E1 6351.62,E2 6351.62} C_VEL
LIN {X 0,Y 123.548,Z 1234.476,A -85,B 0,C 180,E1 6341.882,E2 6341.882} C_VEL
LIN {X 0,Y 135.76,Z 1225.271,A -85,B 0,C 180,E1 6333.674,E2 6333.674} C_VEL
LIN {X 0,Y 149.572,Z 1214.701,A -85,B 0,C 180,E1 6327.246,E2 6327.246} C_VEL
LIN {X 0,Y 165.009,Z 1202.268,A -85,B 0,C 180,E1 6322.019,E2 6322.019} C_VEL
LIN {X 0,Y 180.784,Z 1188.445,A -85,B 0,C 180,E1 6317.964,E2 6317.964} C_VEL
LIN {X 0,Y 195.613,Z 1173.999,A -85,B 0,C 180,E1 6314.977,E2 6314.977} C_VEL
LIN {X 0,Y 211.408,Z 1156.876,A -85,B 0,C 180,E1 6312.415,E2 6312.415} C_VEL
LIN {X 0,Y 225.292,Z 1139.944,A -85,B 0,C 180,E1 6310.58,E2 6310.58} C_VEL
LIN {X 0,Y 238.477,Z 1121.527,A -85,B 0,C 180,E1 6309.125,E2 6309.125} C_VEL
LIN {X 0,Y 250.407,Z 1102.321,A -85,B 0,C 180,E1 6308.021,E2 6308.021} C_VEL
LIN {X 0,Y 261.012,Z 1082.488,A -85,B 0,C 180,E1 6307.197,E2 6307.197} C_VEL
LIN {X 0,Y 270.22,Z 1061.87,A -85,B 0,C 180,E1 6306.556,E2 6306.556} C_VEL
LIN {X 0,Y 277.758,Z 1040.826,A -85,B 0,C 180,E1 6306.018,E2 6306.018} C_VEL
LIN {X 0,Y 284.181,Z 1017.609,A -85,B 0,C 180,E1 6305.521,E2 6305.521} C_VEL
LIN {X 0,Y 288.598,Z 995.208,A -85,B 0,C 180,E1 6305.112,E2 6305.112} C_VEL
LIN {X 0,Y 298.031,Z 915.502,A -85,B 0,C 180,E1 6303.799,E2 6303.799} C_VEL
LIN {X 0,Y 297.775,Z 913.906,A -85,B 0,C 180,E1 6302.694,E2 6302.694} C_VEL
LIN {X 0,Y 297.22,Z 912.672,A -85,B 0,C 180,E1 6298.458,E2 6298.458} C_VEL
LIN {X 0,Y 297.875,Z 914.212,A -85,B 0,C 180,E1 6294.413,E2 6294.413} C_VEL
LIN {X 0,Y 297.932,Z 914.726,A -85,B 0,C 180,E1 6294.116,E2 6294.116} C_VEL
LIN {X 0,Y 291.62,Z 969.508,A -85,B 0,C 180,E1 6293.159,E2 6293.159} C_VEL
LIN {X 0,Y 288.359,Z 992.031,A -85,B 0,C 180,E1 6292.589,E2 6292.589} C_VEL
LIN {X 0,Y 283.538,Z 1013.962,A -85,B 0,C 180,E1 6291.876,E2 6291.876} C_VEL
LIN {X 0,Y 277.348,Z 1034.701,A -85,B 0,C 180,E1 6291.026,E2 6291.026} C_VEL
LIN {X 0,Y 269.546,Z 1054.884,A -85,B 0,C 180,E1 6290.004,E2 6290.004} C_VEL
LIN {X 0,Y 259.972,Z 1075.136,A -85,B 0,C 180,E1 6288.726,E2 6288.726} C_VEL
LIN {X 0,Y 250.032,Z 1092.854,A -85,B 0,C 180,E1 6287.345,E2 6287.345} C_VEL
LIN {X 0,Y 238.413,Z 1110.375,A -85,B 0,C 180,E1 6285.636,E2 6285.636} C_VEL
LIN {X 0,Y 225.794,Z 1126.815,A -85,B 0,C 180,E1 6283.609,E2 6283.609} C_VEL
LIN {X 0,Y 212.317,Z 1142.16,A -85,B 0,C 180,E1 6281.18,E2 6281.18} C_VEL
LIN {X 0,Y 198.084,Z 1156.305,A -85,B 0,C 180,E1 6278.239,E2 6278.239} C_VEL
LIN {X 0,Y 183.563,Z 1168.935,A -85,B 0,C 180,E1 6274.711,E2 6274.711} C_VEL
LIN {X 0,Y 168.257,Z 1180.722,A -85,B 0,C 180,E1 6270.178,E2 6270.178} C_VEL
LIN {X 0,Y 154.06,Z 1190.471,A -85,B 0,C 180,E1 6264.857,E2 6264.857} C_VEL
LIN {X 0,Y 140.63,Z 1198.69,A -85,B 0,C 180,E1 6258.289,E2 6258.289} C_VEL
LIN {X 0,Y 129.112,Z 1205.087,A -85,B 0,C 180,E1 6250.578,E2 6250.578} C_VEL
LIN {X 0,Y 119.597,Z 1210.074,A -85,B 0,C 180,E1 6241.219,E2 6241.219} C_VEL
LIN {X 0,Y 113.053,Z 1213.429,A -85,B 0,C 180,E1 6230.717,E2 6230.717} C_VEL
LIN {X 0,Y 109.673,Z 1215.124,A -85,B 0,C 180,E1 6219.975,E2 6219.975} C_VEL
LIN {X 0,Y 108.801,Z 1215.674,A -85,B 0,C 180,E1 6209.473,E2 6209.473} C_VEL
LIN {X 0,Y 109.764,Z 1215.094,A -85,B 0,C 180,E1 6199.503,E2 6199.503} C_VEL
LIN {X 0,Y 113.248,Z 1213.354,A -85,B 0,C 180,E1 6188.779,E2 6188.779} C_VEL
LIN {X 0,Y 120.061,Z 1209.91,A -85,B 0,C 180,E1 6178.154,E2 6178.154} C_VEL
LIN {X 0,Y 129.545,Z 1204.927,A -85,B 0,C 180,E1 6169.002,E2 6169.002} C_VEL
LIN {X 0,Y 141.777,Z 1198.09,A -85,B 0,C 180,E1 6160.986,E2 6160.986} C_VEL
LIN {X 0,Y 155.345,Z 1189.776,A -85,B 0,C 180,E1 6154.53,E2 6154.53} C_VEL
LIN {X 0,Y 169.712,Z 1179.828,A -85,B 0,C 180,E1 6149.275,E2 6149.275} C_VEL
LIN {X 0,Y 184.271,Z 1168.52,A -85,B 0,C 180,E1 6145.026,E2 6145.026} C_VEL
LIN {X 0,Y 198.829,Z 1155.794,A -85,B 0,C 180,E1 6141.52,E2 6141.52} C_VEL
LIN {X 0,Y 213.097,Z 1141.591,A -85,B 0,C 180,E1 6138.601,E2 6138.601} C_VEL
LIN {X 0,Y 226.462,Z 1126.286,A -85,B 0,C 180,E1 6136.207,E2 6136.207} C_VEL
LIN {X 0,Y 239.68,Z 1108.888,A -85,B 0,C 180,E1 6134.1,E2 6134.1} C_VEL
LIN {X 0,Y 250.873,Z 1091.868,A -85,B 0,C 180,E1 6132.467,E2 6132.467} C_VEL
LIN {X 0,Y 260.827,Z 1073.957,A -85,B 0,C 180,E1 6131.09,E2 6131.09} C_VEL
LIN {X 0,Y 269.954,Z 1054.484,A -85,B 0,C 180,E1 6129.875,E2 6129.875} C_VEL
LIN {X 0,Y 277.531,Z 1034.868,A -85,B 0,C 180,E1 6128.883,E2 6128.883} C_VEL
LIN {X 0,Y 283.851,Z 1013.685,A -85,B 0,C 180,E1 6128.017,E2 6128.017} C_VEL
LIN {X 0,Y 288.611,Z 991.965,A -85,B 0,C 180,E1 6127.314,E2 6127.314} C_VEL
LIN {X 0,Y 291.917,Z 969.013,A -85,B 0,C 180,E1 6126.734,E2 6126.734} C_VEL
LIN {X 0,Y 298.167,Z 914.764,A -85,B 0,C 180,E1 6125.774,E2 6125.774} C_VEL
LIN {X 0,Y 297.861,Z 913.855,A -85,B 0,C 180,E1 6124.621,E2 6124.621} C_VEL
LIN {X 0,Y 297.451,Z 912.996,A -85,B 0,C 180,E1 6120.771,E2 6120.771} C_VEL
LIN {X 0,Y 298.077,Z 914.338,A -85,B 0,C 180,E1 6117.02,E2 6117.02} C_VEL
LIN {X 0,Y 298.254,Z 915.866,A -85,B 0,C 180,E1 6116.154,E2 6116.154} C_VEL
LIN {X 0,Y 288.697,Z 996.178,A -85,B 0,C 180,E1 6114.878,E2 6114.878} C_VEL
LIN {X 0,Y 284.122,Z 1018.867,A -85,B 0,C 180,E1 6114.461,E2 6114.461} C_VEL
LIN {X 0,Y 277.981,Z 1040.827,A -85,B 0,C 180,E1 6113.989,E2 6113.989} C_VEL
LIN {X 0,Y 270.709,Z 1061.237,A -85,B 0,C 180,E1 6113.471,E2 6113.471} C_VEL
LIN {X 0,Y 261.499,Z 1081.915,A -85,B 0,C 180,E1 6112.832,E2 6112.832} C_VEL
LIN {X 0,Y 250.89,Z 1101.844,A -85,B 0,C 180,E1 6112.014,E2 6112.014} C_VEL
LIN {X 0,Y 238.955,Z 1121.126,A -85,B 0,C 180,E1 6110.917,E2 6110.917} C_VEL
LIN {X 0,Y 234.296,Z 1127.916,A -85,B 0,C 180,E1 6110.433,E2 6110.433} C_VEL
LIN {X 0,Y 229.636,Z 1134.05,A -85,B 0,C 180,E1 6110.186,E2 6110.186} C_VEL
LIN {X 0,Y 216.022,Z 1148.872,A -85,B 0,C 180,E1 6110.283,E2 6110.283} C_VEL
LIN {X 0,Y 210.819,Z 1154.455,A -85,B 0,C 180,E1 6109.924,E2 6109.924} C_VEL
LIN {X 0,Y 196.371,Z 1170.01,A -85,B 0,C 180,E1 6107.843,E2 6107.843} C_VEL
LIN {X 0,Y 181.032,Z 1184.673,A -85,B 0,C 180,E1 6105.131,E2 6105.131} C_VEL
LIN {X 0,Y 165.413,Z 1198.137,A -85,B 0,C 180,E1 6101.618,E2 6101.618} C_VEL
LIN {X 0,Y 149.821,Z 1210.443,A -85,B 0,C 180,E1 6097.063,E2 6097.063} C_VEL
LIN {X 0,Y 134.757,Z 1221.394,A -85,B 0,C 180,E1 6091.104,E2 6091.104} C_VEL
LIN {X 0,Y 120.979,Z 1230.979,A -85,B 0,C 180,E1 6083.288,E2 6083.288} C_VEL
LIN {X 0,Y 109.543,Z 1239.125,A -85,B 0,C 180,E1 6073.2,E2 6073.2} C_VEL
LIN {X 0,Y 102.032,Z 1245.421,A -85,B 0,C 180,E1 6061.289,E2 6061.289} C_VEL
LIN {X 0,Y 99.044,Z 1249.605,A -85,B 0,C 180,E1 6048.846,E2 6048.846} C_VEL
LIN {X 0,Y 99.609,Z 1252.025,A -85,B 0,C 180,E1 6037.498,E2 6037.498} C_VEL
LIN {X 0,Y 100.793,Z 1252.658,A -85,B 0,C 180,E1 6030.568,E2 6030.568} C_VEL
LIN {X 0,Y 100.223,Z 1252.375,A -85,B 0,C 180,E1 6025.996,E2 6025.996} C_VEL
LIN {X 0,Y 99.008,Z 1251.021,A -85,B 0,C 180,E1 6017.164,E2 6017.164} C_VEL
LIN {X 0,Y 100.098,Z 1247.574,A -85,B 0,C 180,E1 6004.564,E2 6004.564} C_VEL
LIN {X 0,Y 105.592,Z 1242.203,A -85,B 0,C 180,E1 5992.014,E2 5992.014} C_VEL
LIN {X 0,Y 115.345,Z 1234.871,A -85,B 0,C 180,E1 5981.051,E2 5981.051} C_VEL
